LIN {X 0,Y 331.861,Z 837.829,A -85,B 0,C 180,E1 -14617.89,E2 -14617.89} C_VEL
LIN {X 0,Y 331.677,Z 838.758,A -85,B 0,C 180,E1 -14620.289,E2 -14620.289} C_VEL
LIN {X 0,Y 331.646,Z 838.125,A -85,B 0,C 180,E1 -14622.697,E2 -14622.697} C_VEL
LIN {X 0,Y 331.773,Z 836.768,A -85,B 0,C 180,E1 -14624.35,E2 -14624.35} C_VEL
LIN {X 0,Y 332.117,Z 833.423,A -85,B 0,C 180,E1 -14626.716,E2 -14626.716} C_VEL
LIN {X 0,Y 332.464,Z 829.979,A -85,B 0,C 180,E1 -14628.415,E2 -14628.415} C_VEL
LIN {X 0,Y 332.932,Z 825.524,A -85,B 0,C 180,E1 -14630.123,E2 -14630.123} C_VEL
LIN {X 0,Y 333.677,Z 818.981,A -85,B 0,C 180,E1 -14632.096,E2 -14632.096} C_VEL
LIN {X 0,Y 334.531,Z 811.128,A -85,B 0,C 180,E1 -14633.969,E2 -14633.969} C_VEL
LIN {X 0,Y 335.575,Z 802.763,A -85,B 0,C 180,E1 -14635.567,E2 -14635.567} C_VEL
LIN {X 0,Y 336.737,Z 792.663,A -85,B 0,C 180,E1 -14637.137,E2 -14637.137} C_VEL
LIN {X 0,Y 337.93,Z 781.617,A -85,B 0,C 180,E1 -14638.505,E2 -14638.505} C_VEL
LIN {X 0,Y 339.094,Z 769.813,A -85,B 0,C 180,E1 -14639.657,E2 -14639.657} C_VEL
LIN {X 0,Y 339.897,Z 760.336,A -85,B 0,C 180,E1 -14640.387,E2 -14640.387} C_VEL
LIN {X 0,Y 338.213,Z 747.883,A -85,B 0,C 180,E1 -14641.264,E2 -14641.264} C_VEL
LIN {X 0,Y 335.724,Z 734.171,A -85,B 0,C 180,E1 -14641.988,E2 -14641.988} C_VEL
LIN {X 0,Y 334.799,Z 729.351,A -85,B 0,C 180,E1 -14642.208,E2 -14642.208} C_VEL
LIN {X 0,Y 335.382,Z 720.343,A -85,B 0,C 180,E1 -14645.223,E2 -14645.223} C_VEL
LIN {X 0,Y 336.06,Z 710.471,A -85,B 0,C 180,E1 -14648.533,E2 -14648.533} C_VEL
LIN {X 0,Y 336.777,Z 699.019,A -85,B 0,C 180,E1 -14652.387,E2 -14652.387} C_VEL
LIN {X 0,Y 337.478,Z 687.894,A -85,B 0,C 180,E1 -14656.144,E2 -14656.144} C_VEL
LIN {X 0,Y 337.713,Z 680.208,A -85,B 0,C 180,E1 -14658.774,E2 -14658.774} C_VEL
LIN {X 0,Y 336.611,Z 672.395,A -85,B 0,C 180,E1 -14661.597,E2 -14661.597} C_VEL
LIN {X 0,Y 335.43,Z 665.891,A -85,B 0,C 180,E1 -14663.987,E2 -14663.987} C_VEL
LIN {X 0,Y 333.91,Z 658.899,A -85,B 0,C 180,E1 -14666.682,E2 -14666.682} C_VEL
LIN {X 0,Y 334.089,Z 658.875,A -85,B 0,C 180,E1 -14668.795,E2 -14668.795} C_VEL
LIN {X 0,Y 334.249,Z 658.852,A -85,B 0,C 180,E1 -14670.001,E2 -14670.001} C_VEL
LIN {X 0,Y 334.133,Z 658.866,A -85,B 0,C 180,E1 -14672.412,E2 -14672.412} C_VEL
LIN {X 0,Y 334.014,Z 658.877,A -85,B 0,C 180,E1 -14677.253,E2 -14677.253} C_VEL
LIN {X 0,Y 333.839,Z 658.9,A -85,B 0,C 180,E1 -14680.922,E2 -14680.922} C_VEL
LIN {X 0,Y 333.81,Z 658.906,A -85,B 0,C 180,E1 -14684.635,E2 -14684.635} C_VEL
LIN {X 0,Y 333.799,Z 658.91,A -85,B 0,C 180,E1 -14687.816,E2 -14687.816} C_VEL
LIN {X 0,Y 337.948,Z 672.337,A -85,B 0,C 180,E1 -14689.075,E2 -14689.075} C_VEL
LIN {X 0,Y 340.518,Z 682.415,A -85,B 0,C 180,E1 -14690.207,E2 -14690.207} C_VEL
LIN {X 0,Y 339.514,Z 694.142,A -85,B 0,C 180,E1 -14691.559,E2 -14691.559} C_VEL
LIN {X 0,Y 338.525,Z 704.562,A -85,B 0,C 180,E1 -14693.071,E2 -14693.071} C_VEL
LIN {X 0,Y 337.574,Z 713.136,A -85,B 0,C 180,E1 -14694.607,E2 -14694.607} C_VEL
LIN {X 0,Y 336.576,Z 721.162,A -85,B 0,C 180,E1 -14696.368,E2 -14696.368} C_VEL
LIN {X 0,Y 335.902,Z 726.882,A -85,B 0,C 180,E1 -14697.91,E2 -14697.91} C_VEL
LIN {X 0,Y 335.263,Z 731.79,A -85,B 0,C 180,E1 -14699.514,E2 -14699.514} C_VEL
LIN {X 0,Y 334.713,Z 736.907,A -85,B 0,C 180,E1 -14701.664,E2 -14701.664} C_VEL
LIN {X 0,Y 334.206,Z 740.618,A -85,B 0,C 180,E1 -14703.867,E2 -14703.867} C_VEL
LIN {X 0,Y 333.934,Z 742.948,A -85,B 0,C 180,E1 -14706.107,E2 -14706.107} C_VEL
LIN {X 0,Y 333.914,Z 743.791,A -85,B 0,C 180,E1 -14707.857,E2 -14707.857} C_VEL
LIN {X 0,Y 334.024,Z 743.924,A -85,B 0,C 180,E1 -14709.14,E2 -14709.14} C_VEL
LIN {X 0,Y 334.202,Z 743.41,A -85,B 0,C 180,E1 -14710.795,E2 -14710.795} C_VEL
LIN {X 0,Y 334.556,Z 741.933,A -85,B 0,C 180,E1 -14712.672,E2 -14712.672} C_VEL
LIN {X 0,Y 334.657,Z 741.434,A -85,B 0,C 180,E1 -14713.083,E2 -14713.083} C_VEL
LIN {X 0,Y 334.288,Z 740.325,A -85,B 0,C 180,E1 -14714.071,E2 -14714.071} C_VEL
LIN {X 0,Y 332.022,Z 738.157,A -85,B 0,C 180,E1 -14715.689,E2 -14715.689} C_VEL
LIN {X 0,Y 329.839,Z 735.369,A -85,B 0,C 180,E1 -14717.297,E2 -14717.297} C_VEL
LIN {X 0,Y 329.61,Z 733.111,A -85,B 0,C 180,E1 -14718.253,E2 -14718.253} C_VEL
LIN {X 0,Y 330.871,Z 726.379,A -85,B 0,C 180,E1 -14720.415,E2 -14720.415} C_VEL
LIN {X 0,Y 332.059,Z 719.549,A -85,B 0,C 180,E1 -14722.137,E2 -14722.137} C_VEL
LIN {X 0,Y 333.257,Z 711.36,A -85,B 0,C 180,E1 -14723.809,E2 -14723.809} C_VEL
LIN {X 0,Y 334.746,Z 701.133,A -85,B 0,C 180,E1 -14725.468,E2 -14725.468} C_VEL
LIN {X 0,Y 335.956,Z 690.893,A -85,B 0,C 180,E1 -14726.802,E2 -14726.802} C_VEL
LIN {X 0,Y 336.267,Z 687.695,A -85,B 0,C 180,E1 -14727.159,E2 -14727.159} C_VEL
LIN {X 0,Y 333.454,Z 677.696,A -85,B 0,C 180,E1 -14728.469,E2 -14728.469} C_VEL
LIN {X 0,Y 329.206,Z 666.464,A -85,B 0,C 180,E1 -14729.785,E2 -14729.785} C_VEL
LIN {X 0,Y 326.661,Z 659.793,A -85,B 0,C 180,E1 -14730.474,E2 -14730.474} C_VEL
LIN {X 0,Y 326.691,Z 659.789,A -85,B 0,C 180,E1 -14734.517,E2 -14734.517} C_VEL
LIN {X 0,Y 326.623,Z 659.802,A -85,B 0,C 180,E1 -14738.544,E2 -14738.544} C_VEL
LIN {X 0,Y 326.746,Z 659.786,A -85,B 0,C 180,E1 -14741.178,E2 -14741.178} C_VEL
LIN {X 0,Y 326.765,Z 659.781,A -85,B 0,C 180,E1 -14745.433,E2 -14745.433} C_VEL
LIN {X 0,Y 326.771,Z 659.775,A -85,B 0,C 180,E1 -14748.839,E2 -14748.839} C_VEL
LIN {X 0,Y 326.981,Z 659.745,A -85,B 0,C 180,E1 -14752.591,E2 -14752.591} C_VEL
LIN {X 0,Y 326.78,Z 659.778,A -85,B 0,C 180,E1 -14755.065,E2 -14755.065} C_VEL
LIN {X 0,Y 327.049,Z 659.738,A -85,B 0,C 180,E1 -14757.537,E2 -14757.537} C_VEL
LIN {X 0,Y 327.2,Z 659.721,A -85,B 0,C 180,E1 -14760,E2 -14760} C_VEL
LIN {X 0,Y 327.05,Z 659.746,A -85,B 0,C 180,E1 -14762.463,E2 -14762.463} C_VEL
LIN {X 0,Y 326.998,Z 659.748,A -85,B 0,C 180,E1 -14766.169,E2 -14766.169} C_VEL
LIN {X 0,Y 326.917,Z 659.754,A -85,B 0,C 180,E1 -14768.655,E2 -14768.655} C_VEL
LIN {X 0,Y 326.736,Z 659.779,A -85,B 0,C 180,E1 -14772.421,E2 -14772.421} C_VEL
LIN {X 0,Y 326.756,Z 659.782,A -85,B 0,C 180,E1 -14774.958,E2 -14774.958} C_VEL
LIN {X 0,Y 326.736,Z 659.783,A -85,B 0,C 180,E1 -14778.839,E2 -14778.839} C_VEL
LIN {X 0,Y 326.623,Z 659.794,A -85,B 0,C 180,E1 -14782.787,E2 -14782.787} C_VEL
LIN {X 0,Y 326.692,Z 659.787,A -85,B 0,C 180,E1 -14785.484,E2 -14785.484} C_VEL
LIN {X 0,Y 326.65,Z 659.797,A -85,B 0,C 180,E1 -14789.66,E2 -14789.66} C_VEL
LIN {X 0,Y 326.609,Z 659.805,A -85,B 0,C 180,E1 -14794.019,E2 -14794.019} C_VEL
LIN {X 0,Y 326.63,Z 659.803,A -85,B 0,C 180,E1 -14797.239,E2 -14797.239} C_VEL
LIN {X 0,Y 326.629,Z 659.853,A -85,B 0,C 180,E1 -14800.58,E2 -14800.58} C_VEL
LIN {X 0,Y 328.011,Z 666.445,A -85,B 0,C 180,E1 -14804.135,E2 -14804.135} C_VEL
LIN {X 0,Y 329.365,Z 673.292,A -85,B 0,C 180,E1 -14807.488,E2 -14807.488} C_VEL
LIN {X 0,Y 330.58,Z 679.663,A -85,B 0,C 180,E1 -14810.372,E2 -14810.372} C_VEL
LIN {X 0,Y 331.086,Z 683.496,A -85,B 0,C 180,E1 -14812.005,E2 -14812.005} C_VEL
LIN {X 0,Y 330.051,Z 691.01,A -85,B 0,C 180,E1 -14814.905,E2 -14814.905} C_VEL
LIN {X 0,Y 328.741,Z 701.452,A -85,B 0,C 180,E1 -14818.776,E2 -14818.776} C_VEL
LIN {X 0,Y 327.667,Z 711.906,A -85,B 0,C 180,E1 -14822.538,E2 -14822.538} C_VEL
LIN {X 0,Y 326.622,Z 724.408,A -85,B 0,C 180,E1 -14826.853,E2 -14826.853} C_VEL
LIN {X 0,Y 329.145,Z 739.18,A -85,B 0,C 180,E1 -14827.642,E2 -14827.642} C_VEL
LIN {X 0,Y 330.443,Z 751.644,A -85,B 0,C 180,E1 -14828.469,E2 -14828.469} C_VEL
LIN {X 0,Y 331.025,Z 765.509,A -85,B 0,C 180,E1 -14829.568,E2 -14829.568} C_VEL
LIN {X 0,Y 331.436,Z 777.667,A -85,B 0,C 180,E1 -14830.328,E2 -14830.328} C_VEL
LIN {X 0,Y 331.574,Z 787.793,A -85,B 0,C 180,E1 -14831.141,E2 -14831.141} C_VEL
LIN {X 0,Y 330.277,Z 800.215,A -85,B 0,C 180,E1 -14832.348,E2 -14832.348} C_VEL
LIN {X 0,Y 329.137,Z 811.195,A -85,B 0,C 180,E1 -14833.724,E2 -14833.724} C_VEL
LIN {X 0,Y 328.186,Z 820.112,A -85,B 0,C 180,E1 -14835.109,E2 -14835.109} C_VEL
LIN {X 0,Y 327.013,Z 829.783,A -85,B 0,C 180,E1 -14836.958,E2 -14836.958} C_VEL
LIN {X 0,Y 326.136,Z 837.451,A -85,B 0,C 180,E1 -14838.816,E2 -14838.816} C_VEL
LIN {X 0,Y 325.595,Z 843.592,A -85,B 0,C 180,E1 -14840.683,E2 -14840.683} C_VEL
LIN {X 0,Y 325.224,Z 848.431,A -85,B 0,C 180,E1 -14842.55,E2 -14842.55} C_VEL
LIN {X 0,Y 325.077,Z 851.374,A -85,B 0,C 180,E1 -14843.988,E2 -14843.988} C_VEL
LIN {X 0,Y 324.996,Z 854.734,A -85,B 0,C 180,E1 -14846.28,E2 -14846.28} C_VEL
LIN {X 0,Y 324.927,Z 855.95,A -85,B 0,C 180,E1 -14847.52,E2 -14847.52} C_VEL
LIN {X 0,Y 324.959,Z 856.716,A -85,B 0,C 180,E1 -14848.76,E2 -14848.76} C_VEL
LIN {X 0,Y 325.011,Z 857.06,A -85,B 0,C 180,E1 -14849.999,E2 -14849.999} C_VEL
LIN {X 0,Y 324.942,Z 857.003,A -85,B 0,C 180,E1 -14851.239,E2 -14851.239} C_VEL
LIN {X 0,Y 324.922,Z 856.543,A -85,B 0,C 180,E1 -14852.479,E2 -14852.479} C_VEL
LIN {X 0,Y 324.987,Z 855.631,A -85,B 0,C 180,E1 -14853.719,E2 -14853.719} C_VEL
LIN {X 0,Y 325.018,Z 853.014,A -85,B 0,C 180,E1 -14855.912,E2 -14855.912} C_VEL
LIN {X 0,Y 325.344,Z 849.12,A -85,B 0,C 180,E1 -14858.071,E2 -14858.071} C_VEL
LIN {X 0,Y 325.842,Z 844.566,A -85,B 0,C 180,E1 -14859.935,E2 -14859.935} C_VEL
LIN {X 0,Y 326.665,Z 837.655,A -85,B 0,C 180,E1 -14862.108,E2 -14862.108} C_VEL
LIN {X 0,Y 327.841,Z 830.181,A -85,B 0,C 180,E1 -14863.955,E2 -14863.955} C_VEL
LIN {X 0,Y 328.887,Z 822.723,A -85,B 0,C 180,E1 -14865.465,E2 -14865.465} C_VEL
LIN {X 0,Y 330.233,Z 813.387,A -85,B 0,C 180,E1 -14867.014,E2 -14867.014} C_VEL
LIN {X 0,Y 331.627,Z 803.213,A -85,B 0,C 180,E1 -14868.374,E2 -14868.374} C_VEL
LIN {X 0,Y 333.125,Z 792.076,A -85,B 0,C 180,E1 -14869.567,E2 -14869.567} C_VEL
LIN {X 0,Y 333.537,Z 783.566,A -85,B 0,C 180,E1 -14870.344,E2 -14870.344} C_VEL
LIN {X 0,Y 333.449,Z 770.917,A -85,B 0,C 180,E1 -14871.311,E2 -14871.311} C_VEL
LIN {X 0,Y 332.694,Z 757.681,A -85,B 0,C 180,E1 -14872.083,E2 -14872.083} C_VEL
LIN {X 0,Y 330.545,Z 744.372,A -85,B 0,C 180,E1 -14872.731,E2 -14872.731} C_VEL
LIN {X 0,Y 329.17,Z 737.997,A -85,B 0,C 180,E1 -14873.061,E2 -14873.061} C_VEL
LIN {X 0,Y 327.482,Z 722.292,A -85,B 0,C 180,E1 -14874.907,E2 -14874.907} C_VEL
LIN {X 0,Y 327.209,Z 718.727,A -85,B 0,C 180,E1 -14875.354,E2 -14875.354} C_VEL
LIN {X 0,Y 328.159,Z 708.48,A -85,B 0,C 180,E1 -14878.967,E2 -14878.967} C_VEL
LIN {X 0,Y 329.462,Z 697.365,A -85,B 0,C 180,E1 -14882.952,E2 -14882.952} C_VEL
LIN {X 0,Y 330.775,Z 687.687,A -85,B 0,C 180,E1 -14886.506,E2 -14886.506} C_VEL
LIN {X 0,Y 331.077,Z 683.113,A -85,B 0,C 180,E1 -14888.24,E2 -14888.24} C_VEL
LIN {X 0,Y 330.054,Z 676.875,A -85,B 0,C 180,E1 -14890.768,E2 -14890.768} C_VEL
LIN {X 0,Y 328.431,Z 668.84,A -85,B 0,C 180,E1 -14894.205,E2 -14894.205} C_VEL
LIN {X 0,Y 326.669,Z 659.795,A -85,B 0,C 180,E1 -14898.317,E2 -14898.317} C_VEL
LIN {X 0,Y 326.644,Z 659.797,A -85,B 0,C 180,E1 -14901.394,E2 -14901.394} C_VEL
LIN {X 0,Y 326.616,Z 659.795,A -85,B 0,C 180,E1 -14904.85,E2 -14904.85} C_VEL
LIN {X 0,Y 326.604,Z 659.8,A -85,B 0,C 180,E1 -14907.455,E2 -14907.455} C_VEL
LIN {X 0,Y 326.657,Z 659.794,A -85,B 0,C 180,E1 -14910.34,E2 -14910.34} C_VEL
LIN {X 0,Y 326.686,Z 659.785,A -85,B 0,C 180,E1 -14914.516,E2 -14914.516} C_VEL
LIN {X 0,Y 326.645,Z 659.798,A -85,B 0,C 180,E1 -14918.545,E2 -14918.545} C_VEL
LIN {X 0,Y 326.74,Z 659.787,A -85,B 0,C 180,E1 -14921.177,E2 -14921.177} C_VEL
LIN {X 0,Y 326.758,Z 659.781,A -85,B 0,C 180,E1 -14925.433,E2 -14925.433} C_VEL
LIN {X 0,Y 326.769,Z 659.78,A -85,B 0,C 180,E1 -14928.839,E2 -14928.839} C_VEL
LIN {X 0,Y 326.964,Z 659.839,A -85,B 0,C 180,E1 -14932.071,E2 -14932.071} C_VEL
LIN {X 0,Y 328.395,Z 665.268,A -85,B 0,C 180,E1 -14934.473,E2 -14934.473} C_VEL
LIN {X 0,Y 330.562,Z 672.965,A -85,B 0,C 180,E1 -14937.762,E2 -14937.762} C_VEL
LIN {X 0,Y 331.697,Z 678.579,A -85,B 0,C 180,E1 -14940,E2 -14940} C_VEL
LIN {X 0,Y 332.394,Z 684.908,A -85,B 0,C 180,E1 -14942.423,E2 -14942.423} C_VEL
LIN {X 0,Y 332.288,Z 690.153,A -85,B 0,C 180,E1 -14944.245,E2 -14944.245} C_VEL
LIN {X 0,Y 331.442,Z 699.025,A -85,B 0,C 180,E1 -14947.309,E2 -14947.309} C_VEL
LIN {X 0,Y 330.633,Z 710.037,A -85,B 0,C 180,E1 -14951.029,E2 -14951.029} C_VEL
LIN {X 0,Y 329.691,Z 721.175,A -85,B 0,C 180,E1 -14954.821,E2 -14954.821} C_VEL
LIN {X 0,Y 329.004,Z 730.381,A -85,B 0,C 180,E1 -14957.963,E2 -14957.963} C_VEL
LIN {X 0,Y 332.669,Z 744.629,A -85,B 0,C 180,E1 -14958.874,E2 -14958.874} C_VEL
LIN {X 0,Y 334.735,Z 756.733,A -85,B 0,C 180,E1 -14959.789,E2 -14959.789} C_VEL
LIN {X 0,Y 335.355,Z 762.9,A -85,B 0,C 180,E1 -14960.31,E2 -14960.31} C_VEL
LIN {X 0,Y 334.182,Z 773.988,A -85,B 0,C 180,E1 -14961.24,E2 -14961.24} C_VEL
LIN {X 0,Y 332.896,Z 784.331,A -85,B 0,C 180,E1 -14962.334,E2 -14962.334} C_VEL
LIN {X 0,Y 331.359,Z 795.104,A -85,B 0,C 180,E1 -14963.765,E2 -14963.765} C_VEL
LIN {X 0,Y 330,Z 803.961,A -85,B 0,C 180,E1 -14965.21,E2 -14965.21} C_VEL
LIN {X 0,Y 328.635,Z 812.956,A -85,B 0,C 180,E1 -14967.029,E2 -14967.029} C_VEL
LIN {X 0,Y 327.396,Z 820.622,A -85,B 0,C 180,E1 -14968.983,E2 -14968.983} C_VEL
LIN {X 0,Y 326.65,Z 825.766,A -85,B 0,C 180,E1 -14970.616,E2 -14970.616} C_VEL
LIN {X 0,Y 325.833,Z 831.035,A -85,B 0,C 180,E1 -14972.735,E2 -14972.735} C_VEL
LIN {X 0,Y 325.256,Z 834.796,A -85,B 0,C 180,E1 -14974.808,E2 -14974.808} C_VEL
LIN {X 0,Y 324.882,Z 837.267,A -85,B 0,C 180,E1 -14976.833,E2 -14976.833} C_VEL
LIN {X 0,Y 324.681,Z 838.649,A -85,B 0,C 180,E1 -14978.883,E2 -14978.883} C_VEL
LIN {X 0,Y 324.561,Z 838.967,A -85,B 0,C 180,E1 -14980.724,E2 -14980.724} C_VEL
LIN {X 0,Y 324.544,Z 838.382,A -85,B 0,C 180,E1 -14982.587,E2 -14982.587} C_VEL
LIN {X 0,Y 324.681,Z 836.911,A -85,B 0,C 180,E1 -14984.414,E2 -14984.414} C_VEL
LIN {X 0,Y 324.929,Z 834.578,A -85,B 0,C 180,E1 -14986.202,E2 -14986.202} C_VEL
LIN {X 0,Y 325.274,Z 831.396,A -85,B 0,C 180,E1 -14987.95,E2 -14987.95} C_VEL
LIN {X 0,Y 325.664,Z 827.371,A -85,B 0,C 180,E1 -14989.654,E2 -14989.654} C_VEL
LIN {X 0,Y 326.418,Z 821.17,A -85,B 0,C 180,E1 -14991.711,E2 -14991.711} C_VEL
LIN {X 0,Y 327.195,Z 814.686,A -85,B 0,C 180,E1 -14993.413,E2 -14993.413} C_VEL
LIN {X 0,Y 328.28,Z 806.003,A -85,B 0,C 180,E1 -14995.251,E2 -14995.251} C_VEL
LIN {X 0,Y 329.425,Z 796.379,A -85,B 0,C 180,E1 -14996.895,E2 -14996.895} C_VEL
LIN {X 0,Y 330.744,Z 784.873,A -85,B 0,C 180,E1 -14998.451,E2 -14998.451} C_VEL
LIN {X 0,Y 331.965,Z 772.941,A -85,B 0,C 180,E1 -14999.719,E2 -14999.719} C_VEL
LIN {X 0,Y 333.047,Z 761.183,A -85,B 0,C 180,E1 -15000.68,E2 -15000.68} C_VEL
LIN {X 0,Y 331.507,Z 749.49,A -85,B 0,C 180,E1 -15001.54,E2 -15001.54} C_VEL
LIN {X 0,Y 329.18,Z 736.298,A -85,B 0,C 180,E1 -15002.289,E2 -15002.289} C_VEL
LIN {X 0,Y 327.875,Z 729.497,A -85,B 0,C 180,E1 -15002.602,E2 -15002.602} C_VEL
LIN {X 0,Y 328.521,Z 719.419,A -85,B 0,C 180,E1 -15006.018,E2 -15006.018} C_VEL
LIN {X 0,Y 329.272,Z 709.539,A -85,B 0,C 180,E1 -15009.381,E2 -15009.381} C_VEL
LIN {X 0,Y 329.965,Z 698.474,A -85,B 0,C 180,E1 -15013.146,E2 -15013.146} C_VEL
LIN {X 0,Y 330.589,Z 688.749,A -85,B 0,C 180,E1 -15016.477,E2 -15016.477} C_VEL
LIN {X 0,Y 330.821,Z 681.535,A -85,B 0,C 180,E1 -15018.978,E2 -15018.978} C_VEL
LIN {X 0,Y 329.618,Z 673.201,A -85,B 0,C 180,E1 -15022.034,E2 -15022.034} C_VEL
LIN {X 0,Y 328.353,Z 666.71,A -85,B 0,C 180,E1 -15024.474,E2 -15024.474} C_VEL
LIN {X 0,Y 326.946,Z 659.765,A -85,B 0,C 180,E1 -15027.151,E2 -15027.151} C_VEL
LIN {X 0,Y 327.2,Z 659.729,A -85,B 0,C 180,E1 -15030.001,E2 -15030.001} C_VEL
LIN {X 0,Y 327.069,Z 659.746,A -85,B 0,C 180,E1 -15032.464,E2 -15032.464} C_VEL
LIN {X 0,Y 326.992,Z 659.751,A -85,B 0,C 180,E1 -15036.17,E2 -15036.17} C_VEL
LIN {X 0,Y 326.916,Z 659.764,A -85,B 0,C 180,E1 -15038.656,E2 -15038.656} C_VEL
LIN {X 0,Y 326.74,Z 659.785,A -85,B 0,C 180,E1 -15042.422,E2 -15042.422} C_VEL
LIN {X 0,Y 326.756,Z 659.785,A -85,B 0,C 180,E1 -15044.958,E2 -15044.958} C_VEL
LIN {X 0,Y 326.765,Z 659.96,A -85,B 0,C 180,E1 -15047.444,E2 -15047.444} C_VEL
LIN {X 0,Y 330.61,Z 672.1,A -85,B 0,C 180,E1 -15048.595,E2 -15048.595} C_VEL
LIN {X 0,Y 333.671,Z 683.136,A -85,B 0,C 180,E1 -15049.855,E2 -15049.855} C_VEL
LIN {X 0,Y 332.849,Z 693.349,A -85,B 0,C 180,E1 -15051.036,E2 -15051.036} C_VEL
LIN {X 0,Y 331.82,Z 704.103,A -85,B 0,C 180,E1 -15052.575,E2 -15052.575} C_VEL
LIN {X 0,Y 330.804,Z 713.337,A -85,B 0,C 180,E1 -15054.217,E2 -15054.217} C_VEL
LIN {X 0,Y 329.689,Z 721.838,A -85,B 0,C 180,E1 -15056.095,E2 -15056.095} C_VEL
LIN {X 0,Y 328.804,Z 728.896,A -85,B 0,C 180,E1 -15058.05,E2 -15058.05} C_VEL
LIN {X 0,Y 328.258,Z 733.106,A -85,B 0,C 180,E1 -15059.501,E2 -15059.501} C_VEL
LIN {X 0,Y 327.677,Z 738.165,A -85,B 0,C 180,E1 -15061.7,E2 -15061.7} C_VEL
LIN {X 0,Y 327.172,Z 741.793,A -85,B 0,C 180,E1 -15063.953,E2 -15063.953} C_VEL
LIN {X 0,Y 326.967,Z 743.479,A -85,B 0,C 180,E1 -15065.476,E2 -15065.476} C_VEL
LIN {X 0,Y 326.878,Z 744.654,A -85,B 0,C 180,E1 -15067.296,E2 -15067.296} C_VEL
LIN {X 0,Y 327.014,Z 744.962,A -85,B 0,C 180,E1 -15069.314,E2 -15069.314} C_VEL
LIN {X 0,Y 327.352,Z 743.951,A -85,B 0,C 180,E1 -15071.725,E2 -15071.725} C_VEL
LIN {X 0,Y 327.976,Z 741.402,A -85,B 0,C 180,E1 -15074.141,E2 -15074.141} C_VEL
LIN {X 0,Y 328.544,Z 738.73,A -85,B 0,C 180,E1 -15075.775,E2 -15075.775} C_VEL
LIN {X 0,Y 329.298,Z 735.012,A -85,B 0,C 180,E1 -15077.504,E2 -15077.504} C_VEL
LIN {X 0,Y 329.61,Z 733.111,A -85,B 0,C 180,E1 -15078.253,E2 -15078.253} C_VEL
LIN {X 0,Y 329.429,Z 730.708,A -85,B 0,C 180,E1 -15079.193,E2 -15079.193} C_VEL
LIN {X 0,Y 327.534,Z 726.522,A -85,B 0,C 180,E1 -15080.727,E2 -15080.727} C_VEL
LIN {X 0,Y 325.754,Z 721.651,A -85,B 0,C 180,E1 -15082.207,E2 -15082.207} C_VEL
LIN {X 0,Y 325.739,Z 718.164,A -85,B 0,C 180,E1 -15083.045,E2 -15083.045} C_VEL
LIN {X 0,Y 327.099,Z 709.512,A -85,B 0,C 180,E1 -15084.733,E2 -15084.733} C_VEL
LIN {X 0,Y 328.472,Z 700.088,A -85,B 0,C 180,E1 -15086.2,E2 -15086.2} C_VEL
LIN {X 0,Y 329.624,Z 689.263,A -85,B 0,C 180,E1 -15087.572,E2 -15087.572} C_VEL
LIN {X 0,Y 326.796,Z 679.346,A -85,B 0,C 180,E1 -15088.927,E2 -15088.927} C_VEL
LIN {X 0,Y 323.09,Z 669.418,A -85,B 0,C 180,E1 -15090.16,E2 -15090.16} C_VEL
LIN {X 0,Y 319.683,Z 661.004,A -85,B 0,C 180,E1 -15091.076,E2 -15091.076} C_VEL
LIN {X 0,Y 319.611,Z 660.671,A -85,B 0,C 180,E1 -15091.15,E2 -15091.15} C_VEL
LIN {X 0,Y 319.605,Z 660.675,A -85,B 0,C 180,E1 -15095.304,E2 -15095.304} C_VEL
LIN {X 0,Y 319.606,Z 660.678,A -85,B 0,C 180,E1 -15099.401,E2 -15099.401} C_VEL
LIN {X 0,Y 319.66,Z 660.669,A -85,B 0,C 180,E1 -15102.073,E2 -15102.073} C_VEL
LIN {X 0,Y 319.734,Z 660.657,A -85,B 0,C 180,E1 -15106.008,E2 -15106.008} C_VEL
LIN {X 0,Y 319.76,Z 660.654,A -85,B 0,C 180,E1 -15109.873,E2 -15109.873} C_VEL
LIN {X 0,Y 319.935,Z 660.623,A -85,B 0,C 180,E1 -15112.426,E2 -15112.426} C_VEL
LIN {X 0,Y 319.749,Z 660.654,A -85,B 0,C 180,E1 -15114.956,E2 -15114.956} C_VEL
LIN {X 0,Y 319.993,Z 660.616,A -85,B 0,C 180,E1 -15117.483,E2 -15117.483} C_VEL
LIN {X 0,Y 320.152,Z 660.599,A -85,B 0,C 180,E1 -15120,E2 -15120} C_VEL
LIN {X 0,Y 319.994,Z 660.625,A -85,B 0,C 180,E1 -15122.518,E2 -15122.518} C_VEL
LIN {X 0,Y 319.954,Z 660.627,A -85,B 0,C 180,E1 -15126.306,E2 -15126.306} C_VEL
LIN {X 0,Y 319.845,Z 660.634,A -85,B 0,C 180,E1 -15128.848,E2 -15128.848} C_VEL
LIN {X 0,Y 319.683,Z 660.656,A -85,B 0,C 180,E1 -15132.7,E2 -15132.7} C_VEL
LIN {X 0,Y 319.702,Z 660.66,A -85,B 0,C 180,E1 -15135.296,E2 -15135.296} C_VEL
LIN {X 0,Y 319.677,Z 660.661,A -85,B 0,C 180,E1 -15139.255,E2 -15139.255} C_VEL
LIN {X 0,Y 319.572,Z 660.673,A -85,B 0,C 180,E1 -15143.319,E2 -15143.319} C_VEL
LIN {X 0,Y 319.62,Z 660.668,A -85,B 0,C 180,E1 -15146.09,E2 -15146.09} C_VEL
LIN {X 0,Y 319.582,Z 660.676,A -85,B 0,C 180,E1 -15148.935,E2 -15148.935} C_VEL
LIN {X 0,Y 319.533,Z 660.685,A -85,B 0,C 180,E1 -15151.862,E2 -15151.862} C_VEL
LIN {X 0,Y 319.582,Z 660.68,A -85,B 0,C 180,E1 -15155.543,E2 -15155.543} C_VEL
LIN {X 0,Y 319.561,Z 660.681,A -85,B 0,C 180,E1 -15159.669,E2 -15159.669} C_VEL
LIN {X 0,Y 319.608,Z 660.998,A -85,B 0,C 180,E1 -15160.03,E2 -15160.03} C_VEL
LIN {X 0,Y 321.03,Z 667.662,A -85,B 0,C 180,E1 -15163.743,E2 -15163.743} C_VEL
LIN {X 0,Y 322.241,Z 673.623,A -85,B 0,C 180,E1 -15166.785,E2 -15166.785} C_VEL
LIN {X 0,Y 323.64,Z 681.063,A -85,B 0,C 180,E1 -15170.273,E2 -15170.273} C_VEL
LIN {X 0,Y 324.106,Z 685.046,A -85,B 0,C 180,E1 -15171.989,E2 -15171.989} C_VEL
LIN {X 0,Y 322.806,Z 693.983,A -85,B 0,C 180,E1 -15175.523,E2 -15175.523} C_VEL
LIN {X 0,Y 321.57,Z 703.448,A -85,B 0,C 180,E1 -15179.1,E2 -15179.1} C_VEL
LIN {X 0,Y 320.579,Z 712.936,A -85,B 0,C 180,E1 -15182.588,E2 -15182.588} C_VEL
LIN {X 0,Y 319.667,Z 723.025,A -85,B 0,C 180,E1 -15186.199,E2 -15186.199} C_VEL
LIN {X 0,Y 322.369,Z 738.671,A -85,B 0,C 180,E1 -15187.086,E2 -15187.086} C_VEL
LIN {X 0,Y 323.668,Z 751.03,A -85,B 0,C 180,E1 -15187.951,E2 -15187.951} C_VEL
LIN {X 0,Y 324.164,Z 764.057,A -85,B 0,C 180,E1 -15189.065,E2 -15189.065} C_VEL
LIN {X 0,Y 324.323,Z 770.273,A -85,B 0,C 180,E1 -15189.474,E2 -15189.474} C_VEL
LIN {X 0,Y 324.702,Z 782.978,A -85,B 0,C 180,E1 -15190.397,E2 -15190.397} C_VEL
LIN {X 0,Y 324.537,Z 790.321,A -85,B 0,C 180,E1 -15191.044,E2 -15191.044} C_VEL
LIN {X 0,Y 323.319,Z 800.819,A -85,B 0,C 180,E1 -15192.119,E2 -15192.119} C_VEL
LIN {X 0,Y 322.143,Z 811.603,A -85,B 0,C 180,E1 -15193.523,E2 -15193.523} C_VEL
LIN {X 0,Y 321.054,Z 821.311,A -85,B 0,C 180,E1 -15195.095,E2 -15195.095} C_VEL
LIN {X 0,Y 320.074,Z 829.268,A -85,B 0,C 180,E1 -15196.67,E2 -15196.67} C_VEL
LIN {X 0,Y 319.114,Z 837.012,A -85,B 0,C 180,E1 -15198.567,E2 -15198.567} C_VEL
LIN {X 0,Y 318.551,Z 843.2,A -85,B 0,C 180,E1 -15200.475,E2 -15200.475} C_VEL
LIN {X 0,Y 318.177,Z 848.081,A -85,B 0,C 180,E1 -15202.384,E2 -15202.384} C_VEL
LIN {X 0,Y 317.97,Z 851.405,A -85,B 0,C 180,E1 -15204.057,E2 -15204.057} C_VEL
LIN {X 0,Y 317.902,Z 854.458,A -85,B 0,C 180,E1 -15206.197,E2 -15206.197} C_VEL
LIN {X 0,Y 317.846,Z 855.692,A -85,B 0,C 180,E1 -15207.465,E2 -15207.465} C_VEL
LIN {X 0,Y 317.864,Z 856.49,A -85,B 0,C 180,E1 -15208.732,E2 -15208.732} C_VEL
LIN {X 0,Y 317.913,Z 856.85,A -85,B 0,C 180,E1 -15209.999,E2 -15209.999} C_VEL
LIN {X 0,Y 317.848,Z 856.809,A -85,B 0,C 180,E1 -15211.266,E2 -15211.266} C_VEL
LIN {X 0,Y 317.841,Z 856.372,A -85,B 0,C 180,E1 -15212.534,E2 -15212.534} C_VEL
LIN {X 0,Y 317.892,Z 855.49,A -85,B 0,C 180,E1 -15213.802,E2 -15213.802} C_VEL
LIN {X 0,Y 317.923,Z 853.182,A -85,B 0,C 180,E1 -15215.86,E2 -15215.86} C_VEL
LIN {X 0,Y 318.284,Z 849.059,A -85,B 0,C 180,E1 -15218.251,E2 -15218.251} C_VEL
LIN {X 0,Y 318.835,Z 844.546,A -85,B 0,C 180,E1 -15220.156,E2 -15220.156} C_VEL
LIN {X 0,Y 319.712,Z 837.702,A -85,B 0,C 180,E1 -15222.375,E2 -15222.375} C_VEL
LIN {X 0,Y 320.934,Z 830.278,A -85,B 0,C 180,E1 -15224.261,E2 -15224.261} C_VEL
LIN {X 0,Y 322.134,Z 821.985,A -85,B 0,C 180,E1 -15225.983,E2 -15225.983} C_VEL
LIN {X 0,Y 323.569,Z 812.681,A -85,B 0,C 180,E1 -15227.539,E2 -15227.539} C_VEL
LIN {X 0,Y 325.071,Z 802.452,A -85,B 0,C 180,E1 -15228.922,E2 -15228.922} C_VEL
LIN {X 0,Y 326.635,Z 791.209,A -85,B 0,C 180,E1 -15230.136,E2 -15230.136} C_VEL
LIN {X 0,Y 326.929,Z 782.576,A -85,B 0,C 180,E1 -15230.939,E2 -15230.939} C_VEL
LIN {X 0,Y 326.907,Z 770.404,A -85,B 0,C 180,E1 -15231.878,E2 -15231.878} C_VEL
LIN {X 0,Y 326.202,Z 757.985,A -85,B 0,C 180,E1 -15232.628,E2 -15232.628} C_VEL
LIN {X 0,Y 324.093,Z 745.01,A -85,B 0,C 180,E1 -15233.303,E2 -15233.303} C_VEL
LIN {X 0,Y 322.568,Z 737.897,A -85,B 0,C 180,E1 -15233.685,E2 -15233.685} C_VEL
LIN {X 0,Y 320.898,Z 720.964,A -85,B 0,C 180,E1 -15235.802,E2 -15235.802} C_VEL
LIN {X 0,Y 320.397,Z 715.96,A -85,B 0,C 180,E1 -15236.528,E2 -15236.528} C_VEL
LIN {X 0,Y 321.458,Z 705.881,A -85,B 0,C 180,E1 -15240.187,E2 -15240.187} C_VEL
LIN {X 0,Y 322.802,Z 695.115,A -85,B 0,C 180,E1 -15244.174,E2 -15244.174} C_VEL
LIN {X 0,Y 324.025,Z 686.58,A -85,B 0,C 180,E1 -15247.394,E2 -15247.394} C_VEL
LIN {X 0,Y 323.992,Z 683.388,A -85,B 0,C 180,E1 -15248.656,E2 -15248.656} C_VEL
LIN {X 0,Y 322.795,Z 676.712,A -85,B 0,C 180,E1 -15251.458,E2 -15251.458} C_VEL
LIN {X 0,Y 321.213,Z 668.768,A -85,B 0,C 180,E1 -15254.96,E2 -15254.96} C_VEL
LIN {X 0,Y 319.622,Z 660.674,A -85,B 0,C 180,E1 -15258.779,E2 -15258.779} C_VEL
LIN {X 0,Y 319.58,Z 660.67,A -85,B 0,C 180,E1 -15262.342,E2 -15262.342} C_VEL
LIN {X 0,Y 319.556,Z 660.672,A -85,B 0,C 180,E1 -15265.123,E2 -15265.123} C_VEL
LIN {X 0,Y 319.566,Z 660.673,A -85,B 0,C 180,E1 -15269.057,E2 -15269.057} C_VEL
LIN {X 0,Y 319.605,Z 660.674,A -85,B 0,C 180,E1 -15272.498,E2 -15272.498} C_VEL
LIN {X 0,Y 319.601,Z 660.672,A -85,B 0,C 180,E1 -15275.303,E2 -15275.303} C_VEL
LIN {X 0,Y 319.593,Z 660.674,A -85,B 0,C 180,E1 -15278.047,E2 -15278.047} C_VEL
LIN {X 0,Y 319.685,Z 660.664,A -85,B 0,C 180,E1 -15280.961,E2 -15280.961} C_VEL
LIN {X 0,Y 319.726,Z 660.656,A -85,B 0,C 180,E1 -15285.275,E2 -15285.275} C_VEL
LIN {X 0,Y 319.755,Z 660.655,A -85,B 0,C 180,E1 -15289.873,E2 -15289.873} C_VEL
LIN {X 0,Y 319.849,Z 660.824,A -85,B 0,C 180,E1 -15290.833,E2 -15290.833} C_VEL
LIN {X 0,Y 321.765,Z 666.854,A -85,B 0,C 180,E1 -15293.73,E2 -15293.73} C_VEL
LIN {X 0,Y 324.013,Z 675.44,A -85,B 0,C 180,E1 -15297.513,E2 -15297.513} C_VEL
LIN {X 0,Y 325.168,Z 681.464,A -85,B 0,C 180,E1 -15300,E2 -15300} C_VEL
LIN {X 0,Y 325.763,Z 686.259,A -85,B 0,C 180,E1 -15301.854,E2 -15301.854} C_VEL
LIN {X 0,Y 325.666,Z 691.21,A -85,B 0,C 180,E1 -15303.712,E2 -15303.712} C_VEL
LIN {X 0,Y 324.834,Z 700.298,A -85,B 0,C 180,E1 -15306.834,E2 -15306.834} C_VEL
LIN {X 0,Y 323.892,Z 711.232,A -85,B 0,C 180,E1 -15310.628,E2 -15310.628} C_VEL
LIN {X 0,Y 323.082,Z 720.501,A -85,B 0,C 180,E1 -15313.844,E2 -15313.844} C_VEL
LIN {X 0,Y 322.241,Z 730.553,A -85,B 0,C 180,E1 -15317.327,E2 -15317.327} C_VEL
LIN {X 0,Y 325.909,Z 744.508,A -85,B 0,C 180,E1 -15318.262,E2 -15318.262} C_VEL
LIN {X 0,Y 327.909,Z 755.347,A -85,B 0,C 180,E1 -15319.11,E2 -15319.11} C_VEL
LIN {X 0,Y 328.821,Z 764.222,A -85,B 0,C 180,E1 -15319.88,E2 -15319.88} C_VEL
LIN {X 0,Y 327.51,Z 775.797,A -85,B 0,C 180,E1 -15320.901,E2 -15320.901} C_VEL
LIN {X 0,Y 325.974,Z 786.926,A -85,B 0,C 180,E1 -15322.153,E2 -15322.153} C_VEL
LIN {X 0,Y 324.416,Z 797.383,A -85,B 0,C 180,E1 -15323.627,E2 -15323.627} C_VEL
LIN {X 0,Y 323.032,Z 805.857,A -85,B 0,C 180,E1 -15325.103,E2 -15325.103} C_VEL
LIN {X 0,Y 321.693,Z 814.012,A -85,B 0,C 180,E1 -15326.851,E2 -15326.851} C_VEL
LIN {X 0,Y 320.395,Z 821.542,A -85,B 0,C 180,E1 -15328.854,E2 -15328.854} C_VEL
LIN {X 0,Y 319.446,Z 827.582,A -85,B 0,C 180,E1 -15330.907,E2 -15330.907} C_VEL
LIN {X 0,Y 318.66,Z 832.395,A -85,B 0,C 180,E1 -15333.064,E2 -15333.064} C_VEL
LIN {X 0,Y 318.092,Z 835.787,A -85,B 0,C 180,E1 -15335.168,E2 -15335.168} C_VEL
LIN {X 0,Y 317.753,Z 837.956,A -85,B 0,C 180,E1 -15337.229,E2 -15337.229} C_VEL
LIN {X 0,Y 317.554,Z 839.022,A -85,B 0,C 180,E1 -15339.232,E2 -15339.232} C_VEL
LIN {X 0,Y 317.44,Z 838.982,A -85,B 0,C 180,E1 -15341.62,E2 -15341.62} C_VEL
LIN {X 0,Y 317.49,Z 838.073,A -85,B 0,C 180,E1 -15343.331,E2 -15343.331} C_VEL
LIN {X 0,Y 317.792,Z 835.26,A -85,B 0,C 180,E1 -15345.905,E2 -15345.905} C_VEL
LIN {X 0,Y 318.132,Z 832.278,A -85,B 0,C 180,E1 -15347.684,E2 -15347.684} C_VEL
LIN {X 0,Y 318.642,Z 827.361,A -85,B 0,C 180,E1 -15349.855,E2 -15349.855} C_VEL
LIN {X 0,Y 319.428,Z 821.026,A -85,B 0,C 180,E1 -15351.973,E2 -15351.973} C_VEL
LIN {X 0,Y 320.379,Z 813.277,A -85,B 0,C 180,E1 -15353.992,E2 -15353.992} C_VEL
LIN {X 0,Y 321.496,Z 804.733,A -85,B 0,C 180,E1 -15355.776,E2 -15355.776} C_VEL
LIN {X 0,Y 322.579,Z 796.015,A -85,B 0,C 180,E1 -15357.254,E2 -15357.254} C_VEL
LIN {X 0,Y 323.89,Z 784.928,A -85,B 0,C 180,E1 -15358.774,E2 -15358.774} C_VEL
LIN {X 0,Y 325.063,Z 773.86,A -85,B 0,C 180,E1 -15359.985,E2 -15359.985} C_VEL
LIN {X 0,Y 326.215,Z 761.749,A -85,B 0,C 180,E1 -15361.005,E2 -15361.005} C_VEL
LIN {X 0,Y 324.438,Z 748.768,A -85,B 0,C 180,E1 -15361.98,E2 -15361.98} C_VEL
LIN {X 0,Y 322.062,Z 735.536,A -85,B 0,C 180,E1 -15362.726,E2 -15362.726} C_VEL
LIN {X 0,Y 320.959,Z 729.669,A -85,B 0,C 180,E1 -15362.994,E2 -15362.994} C_VEL
LIN {X 0,Y 321.738,Z 718.473,A -85,B 0,C 180,E1 -15366.848,E2 -15366.848} C_VEL
LIN {X 0,Y 322.445,Z 708.473,A -85,B 0,C 180,E1 -15370.287,E2 -15370.287} C_VEL
LIN {X 0,Y 323.062,Z 698.978,A -85,B 0,C 180,E1 -15373.573,E2 -15373.573} C_VEL
LIN {X 0,Y 323.718,Z 689.595,A -85,B 0,C 180,E1 -15376.824,E2 -15376.824} C_VEL
LIN {X 0,Y 323.964,Z 684.119,A -85,B 0,C 180,E1 -15378.742,E2 -15378.742} C_VEL
LIN {X 0,Y 323.146,Z 677.34,A -85,B 0,C 180,E1 -15381.244,E2 -15381.244} C_VEL
LIN {X 0,Y 321.997,Z 670.757,A -85,B 0,C 180,E1 -15383.735,E2 -15383.735} C_VEL
LIN {X 0,Y 320.007,Z 660.627,A -85,B 0,C 180,E1 -15387.719,E2 -15387.719} C_VEL
LIN {X 0,Y 320.152,Z 660.607,A -85,B 0,C 180,E1 -15390.001,E2 -15390.001} C_VEL
LIN {X 0,Y 320.01,Z 660.625,A -85,B 0,C 180,E1 -15392.518,E2 -15392.518} C_VEL
LIN {X 0,Y 319.947,Z 660.627,A -85,B 0,C 180,E1 -15396.306,E2 -15396.306} C_VEL
LIN {X 0,Y 319.844,Z 660.643,A -85,B 0,C 180,E1 -15398.849,E2 -15398.849} C_VEL
LIN {X 0,Y 319.687,Z 660.664,A -85,B 0,C 180,E1 -15402.7,E2 -15402.7} C_VEL
LIN {X 0,Y 319.701,Z 660.664,A -85,B 0,C 180,E1 -15405.296,E2 -15405.296} C_VEL
LIN {X 0,Y 319.691,Z 660.72,A -85,B 0,C 180,E1 -15407.018,E2 -15407.018} C_VEL
LIN {X 0,Y 323.54,Z 672.841,A -85,B 0,C 180,E1 -15408.196,E2 -15408.196} C_VEL
LIN {X 0,Y 326.629,Z 683.871,A -85,B 0,C 180,E1 -15409.482,E2 -15409.482} C_VEL
LIN {X 0,Y 326.883,Z 685.01,A -85,B 0,C 180,E1 -15409.63,E2 -15409.63} C_VEL
LIN {X 0,Y 325.859,Z 696.429,A -85,B 0,C 180,E1 -15411.012,E2 -15411.012} C_VEL
LIN {X 0,Y 324.891,Z 705.895,A -85,B 0,C 180,E1 -15412.433,E2 -15412.433} C_VEL
LIN {X 0,Y 323.723,Z 715.607,A -85,B 0,C 180,E1 -15414.243,E2 -15414.243} C_VEL
LIN {X 0,Y 322.592,Z 724.145,A -85,B 0,C 180,E1 -15416.226,E2 -15416.226} C_VEL
LIN {X 0,Y 321.657,Z 731.337,A -85,B 0,C 180,E1 -15418.374,E2 -15418.374} C_VEL
LIN {X 0,Y 321.027,Z 736.227,A -85,B 0,C 180,E1 -15420.234,E2 -15420.234} C_VEL
LIN {X 0,Y 320.441,Z 740.752,A -85,B 0,C 180,E1 -15422.503,E2 -15422.503} C_VEL
LIN {X 0,Y 320.017,Z 743.859,A -85,B 0,C 180,E1 -15424.82,E2 -15424.82} C_VEL
LIN {X 0,Y 319.877,Z 745.189,A -85,B 0,C 180,E1 -15426.386,E2 -15426.386} C_VEL
LIN {X 0,Y 319.888,Z 745.881,A -85,B 0,C 180,E1 -15427.964,E2 -15427.964} C_VEL
LIN {X 0,Y 320.062,Z 745.938,A -85,B 0,C 180,E1 -15429.777,E2 -15429.777} C_VEL
LIN {X 0,Y 320.359,Z 745.067,A -85,B 0,C 180,E1 -15431.765,E2 -15431.765} C_VEL
LIN {X 0,Y 320.826,Z 743.254,A -85,B 0,C 180,E1 -15433.706,E2 -15433.706} C_VEL
LIN {X 0,Y 321.695,Z 739.538,A -85,B 0,C 180,E1 -15436.133,E2 -15436.133} C_VEL
LIN {X 0,Y 322.452,Z 735.943,A -85,B 0,C 180,E1 -15437.821,E2 -15437.821} C_VEL
LIN {X 0,Y 323.568,Z 730.197,A -85,B 0,C 180,E1 -15439.913,E2 -15439.913} C_VEL
LIN {X 0,Y 324.704,Z 723.992,A -85,B 0,C 180,E1 -15441.685,E2 -15441.685} C_VEL
LIN {X 0,Y 325.739,Z 718.164,A -85,B 0,C 180,E1 -15443.045,E2 -15443.045} C_VEL
LIN {X 0,Y 325.722,Z 714.517,A -85,B 0,C 180,E1 -15443.861,E2 -15443.861} C_VEL
LIN {X 0,Y 324.007,Z 708.442,A -85,B 0,C 180,E1 -15445.216,E2 -15445.216} C_VEL
LIN {X 0,Y 322.378,Z 701.882,A -85,B 0,C 180,E1 -15446.499,E2 -15446.499} C_VEL
LIN {X 0,Y 322.448,Z 697.377,A -85,B 0,C 180,E1 -15447.177,E2 -15447.177} C_VEL
LIN {X 0,Y 323.09,Z 691.845,A -85,B 0,C 180,E1 -15447.87,E2 -15447.87} C_VEL
LIN {X 0,Y 320.689,Z 682.667,A -85,B 0,C 180,E1 -15449.185,E2 -15449.185} C_VEL
LIN {X 0,Y 316.752,Z 671.846,A -85,B 0,C 180,E1 -15450.6,E2 -15450.6} C_VEL
LIN {X 0,Y 312.642,Z 661.964,A -85,B 0,C 180,E1 -15451.752,E2 -15451.752} C_VEL
LIN {X 0,Y 312.587,Z 661.551,A -85,B 0,C 180,E1 -15451.826,E2 -15451.826} C_VEL
LIN {X 0,Y 312.586,Z 661.547,A -85,B 0,C 180,E1 -15454.711,E2 -15454.711} C_VEL
LIN {X 0,Y 312.541,Z 661.556,A -85,B 0,C 180,E1 -15458.913,E2 -15458.913} C_VEL
LIN {X 0,Y 312.64,Z 661.547,A -85,B 0,C 180,E1 -15461.657,E2 -15461.657} C_VEL
LIN {X 0,Y 312.696,Z 661.533,A -85,B 0,C 180,E1 -15465.686,E2 -15465.686} C_VEL
LIN {X 0,Y 312.704,Z 661.53,A -85,B 0,C 180,E1 -15469.642,E2 -15469.642} C_VEL
LIN {X 0,Y 312.874,Z 661.503,A -85,B 0,C 180,E1 -15472.254,E2 -15472.254} C_VEL
LIN {X 0,Y 312.72,Z 661.529,A -85,B 0,C 180,E1 -15474.843,E2 -15474.843} C_VEL
LIN {X 0,Y 312.993,Z 661.496,A -85,B 0,C 180,E1 -15478.714,E2 -15478.714} C_VEL
LIN {X 0,Y 312.993,Z 661.486,A -85,B 0,C 180,E1 -15481.287,E2 -15481.287} C_VEL
LIN {X 0,Y 312.72,Z 661.519,A -85,B 0,C 180,E1 -15485.158,E2 -15485.158} C_VEL
LIN {X 0,Y 312.874,Z 661.512,A -85,B 0,C 180,E1 -15487.746,E2 -15487.746} C_VEL
LIN {X 0,Y 312.671,Z 661.538,A -85,B 0,C 180,E1 -15491.671,E2 -15491.671} C_VEL
LIN {X 0,Y 312.702,Z 661.533,A -85,B 0,C 180,E1 -15494.888,E2 -15494.888} C_VEL
LIN {X 0,Y 312.633,Z 661.538,A -85,B 0,C 180,E1 -15499.237,E2 -15499.237} C_VEL
LIN {X 0,Y 312.548,Z 661.547,A -85,B 0,C 180,E1 -15502.789,E2 -15502.789} C_VEL
LIN {X 0,Y 312.599,Z 661.542,A -85,B 0,C 180,E1 -15505.933,E2 -15505.933} C_VEL
LIN {X 0,Y 312.54,Z 661.554,A -85,B 0,C 180,E1 -15509.651,E2 -15509.651} C_VEL
LIN {X 0,Y 312.522,Z 661.559,A -85,B 0,C 180,E1 -15513.689,E2 -15513.689} C_VEL
LIN {X 0,Y 312.523,Z 661.561,A -85,B 0,C 180,E1 -15517.386,E2 -15517.386} C_VEL
LIN {X 0,Y 312.509,Z 661.716,A -85,B 0,C 180,E1 -15519.182,E2 -15519.182} C_VEL
LIN {X 0,Y 313.965,Z 668.318,A -85,B 0,C 180,E1 -15523.057,E2 -15523.057} C_VEL
LIN {X 0,Y 315.354,Z 675.237,A -85,B 0,C 180,E1 -15526.695,E2 -15526.695} C_VEL
LIN {X 0,Y 316.809,Z 683.219,A -85,B 0,C 180,E1 -15530.497,E2 -15530.497} C_VEL
LIN {X 0,Y 317.122,Z 685.756,A -85,B 0,C 180,E1 -15531.645,E2 -15531.645} C_VEL
LIN {X 0,Y 316.384,Z 691.362,A -85,B 0,C 180,E1 -15533.938,E2 -15533.938} C_VEL
LIN {X 0,Y 314.896,Z 701.748,A -85,B 0,C 180,E1 -15538.006,E2 -15538.006} C_VEL
LIN {X 0,Y 313.702,Z 712.078,A -85,B 0,C 180,E1 -15541.935,E2 -15541.935} C_VEL
LIN {X 0,Y 312.737,Z 721.812,A -85,B 0,C 180,E1 -15545.527,E2 -15545.527} C_VEL
LIN {X 0,Y 315.626,Z 738.173,A -85,B 0,C 180,E1 -15546.508,E2 -15546.508} C_VEL
LIN {X 0,Y 317.002,Z 751.495,A -85,B 0,C 180,E1 -15547.496,E2 -15547.496} C_VEL
LIN {X 0,Y 317.427,Z 764.719,A -85,B 0,C 180,E1 -15548.685,E2 -15548.685} C_VEL
LIN {X 0,Y 317.449,Z 767.949,A -85,B 0,C 180,E1 -15548.97,E2 -15548.97} C_VEL
LIN {X 0,Y 317.767,Z 780.727,A -85,B 0,C 180,E1 -15549.867,E2 -15549.867} C_VEL
LIN {X 0,Y 317.751,Z 789.262,A -85,B 0,C 180,E1 -15550.623,E2 -15550.623} C_VEL
LIN {X 0,Y 316.363,Z 801.283,A -85,B 0,C 180,E1 -15551.879,E2 -15551.879} C_VEL
LIN {X 0,Y 315.104,Z 812.611,A -85,B 0,C 180,E1 -15553.417,E2 -15553.417} C_VEL
LIN {X 0,Y 313.916,Z 822.425,A -85,B 0,C 180,E1 -15555.08,E2 -15555.08} C_VEL
LIN {X 0,Y 312.738,Z 831.489,A -85,B 0,C 180,E1 -15557.013,E2 -15557.013} C_VEL
LIN {X 0,Y 311.917,Z 838.78,A -85,B 0,C 180,E1 -15558.958,E2 -15558.958} C_VEL
LIN {X 0,Y 311.358,Z 844.579,A -85,B 0,C 180,E1 -15560.908,E2 -15560.908} C_VEL
LIN {X 0,Y 311.013,Z 849.099,A -85,B 0,C 180,E1 -15562.86,E2 -15562.86} C_VEL
LIN {X 0,Y 310.836,Z 852.495,A -85,B 0,C 180,E1 -15564.81,E2 -15564.81} C_VEL
LIN {X 0,Y 310.81,Z 854.167,A -85,B 0,C 180,E1 -15566.11,E2 -15566.11} C_VEL
LIN {X 0,Y 310.766,Z 855.42,A -85,B 0,C 180,E1 -15567.407,E2 -15567.407} C_VEL
LIN {X 0,Y 310.772,Z 856.256,A -85,B 0,C 180,E1 -15568.703,E2 -15568.703} C_VEL
LIN {X 0,Y 310.818,Z 856.638,A -85,B 0,C 180,E1 -15569.999,E2 -15569.999} C_VEL
LIN {X 0,Y 310.757,Z 856.617,A -85,B 0,C 180,E1 -15571.295,E2 -15571.295} C_VEL
LIN {X 0,Y 310.761,Z 856.199,A -85,B 0,C 180,E1 -15572.592,E2 -15572.592} C_VEL
LIN {X 0,Y 310.799,Z 855.355,A -85,B 0,C 180,E1 -15573.889,E2 -15573.889} C_VEL
LIN {X 0,Y 310.84,Z 853.317,A -85,B 0,C 180,E1 -15575.827,E2 -15575.827} C_VEL
LIN {X 0,Y 311.096,Z 850.262,A -85,B 0,C 180,E1 -15577.789,E2 -15577.789} C_VEL
LIN {X 0,Y 311.619,Z 846.163,A -85,B 0,C 180,E1 -15579.738,E2 -15579.738} C_VEL
LIN {X 0,Y 312.454,Z 839.884,A -85,B 0,C 180,E1 -15582.008,E2 -15582.008} C_VEL
LIN {X 0,Y 313.608,Z 833.073,A -85,B 0,C 180,E1 -15583.939,E2 -15583.939} C_VEL
LIN {X 0,Y 314.961,Z 824.944,A -85,B 0,C 180,E1 -15585.796,E2 -15585.796} C_VEL
LIN {X 0,Y 316.385,Z 815.972,A -85,B 0,C 180,E1 -15587.449,E2 -15587.449} C_VEL
LIN {X 0,Y 318.014,Z 805.39,A -85,B 0,C 180,E1 -15589.023,E2 -15589.023} C_VEL
LIN {X 0,Y 319.654,Z 794.9,A -85,B 0,C 180,E1 -15590.259,E2 -15590.259} C_VEL
LIN {X 0,Y 320.361,Z 786.994,A -85,B 0,C 180,E1 -15591.052,E2 -15591.052} C_VEL
LIN {X 0,Y 320.486,Z 774.62,A -85,B 0,C 180,E1 -15592.131,E2 -15592.131} C_VEL
LIN {X 0,Y 320.038,Z 760.917,A -85,B 0,C 180,E1 -15593.05,E2 -15593.05} C_VEL
LIN {X 0,Y 318.298,Z 748.588,A -85,B 0,C 180,E1 -15593.748,E2 -15593.748} C_VEL
LIN {X 0,Y 315.968,Z 737.511,A -85,B 0,C 180,E1 -15594.385,E2 -15594.385} C_VEL
LIN {X 0,Y 314.654,Z 723.363,A -85,B 0,C 180,E1 -15596.243,E2 -15596.243} C_VEL
LIN {X 0,Y 313.652,Z 713.162,A -85,B 0,C 180,E1 -15597.769,E2 -15597.769} C_VEL
LIN {X 0,Y 314.982,Z 701.844,A -85,B 0,C 180,E1 -15602.019,E2 -15602.019} C_VEL
LIN {X 0,Y 316.472,Z 691.282,A -85,B 0,C 180,E1 -15606.049,E2 -15606.049} C_VEL
LIN {X 0,Y 317.052,Z 687.282,A -85,B 0,C 180,E1 -15607.609,E2 -15607.609} C_VEL
LIN {X 0,Y 316.911,Z 683.674,A -85,B 0,C 180,E1 -15609.087,E2 -15609.087} C_VEL
LIN {X 0,Y 315.314,Z 675.463,A -85,B 0,C 180,E1 -15612.647,E2 -15612.647} C_VEL
LIN {X 0,Y 313.83,Z 668.079,A -85,B 0,C 180,E1 -15616.034,E2 -15616.034} C_VEL
LIN {X 0,Y 312.56,Z 661.552,A -85,B 0,C 180,E1 -15619.195,E2 -15619.195} C_VEL
LIN {X 0,Y 312.538,Z 661.547,A -85,B 0,C 180,E1 -15622.616,E2 -15622.616} C_VEL
LIN {X 0,Y 312.516,Z 661.553,A -85,B 0,C 180,E1 -15626.31,E2 -15626.31} C_VEL
LIN {X 0,Y 312.541,Z 661.552,A -85,B 0,C 180,E1 -15630.349,E2 -15630.349} C_VEL
LIN {X 0,Y 312.599,Z 661.539,A -85,B 0,C 180,E1 -15634.064,E2 -15634.064} C_VEL
LIN {X 0,Y 312.583,Z 661.543,A -85,B 0,C 180,E1 -15637.528,E2 -15637.528} C_VEL
LIN {X 0,Y 312.634,Z 661.541,A -85,B 0,C 180,E1 -15641.656,E2 -15641.656} C_VEL
LIN {X 0,Y 312.689,Z 661.535,A -85,B 0,C 180,E1 -15645.686,E2 -15645.686} C_VEL
LIN {X 0,Y 312.704,Z 661.566,A -85,B 0,C 180,E1 -15649.314,E2 -15649.314} C_VEL
LIN {X 0,Y 315.05,Z 668.616,A -85,B 0,C 180,E1 -15652.952,E2 -15652.952} C_VEL
LIN {X 0,Y 317.582,Z 678.468,A -85,B 0,C 180,E1 -15657.463,E2 -15657.463} C_VEL
LIN {X 0,Y 318.694,Z 684.462,A -85,B 0,C 180,E1 -15660,E2 -15660} C_VEL
LIN {X 0,Y 319.167,Z 689.176,A -85,B 0,C 180,E1 -15661.893,E2 -15661.893} C_VEL
LIN {X 0,Y 318.977,Z 694.354,A -85,B 0,C 180,E1 -15663.79,E2 -15663.79} C_VEL
LIN {X 0,Y 318.063,Z 703.36,A -85,B 0,C 180,E1 -15666.98,E2 -15666.98} C_VEL
LIN {X 0,Y 317.048,Z 714.314,A -85,B 0,C 180,E1 -15670.86,E2 -15670.86} C_VEL
LIN {X 0,Y 315.968,Z 725.556,A -85,B 0,C 180,E1 -15674.82,E2 -15674.82} C_VEL
LIN {X 0,Y 315.535,Z 730.766,A -85,B 0,C 180,E1 -15676.665,E2 -15676.665} C_VEL
LIN {X 0,Y 319.332,Z 744.897,A -85,B 0,C 180,E1 -15677.656,E2 -15677.656} C_VEL
LIN {X 0,Y 321.422,Z 756.299,A -85,B 0,C 180,E1 -15678.587,E2 -15678.587} C_VEL
LIN {X 0,Y 322.253,Z 765.937,A -85,B 0,C 180,E1 -15679.459,E2 -15679.459} C_VEL
LIN {X 0,Y 320.859,Z 777.273,A -85,B 0,C 180,E1 -15680.515,E2 -15680.515} C_VEL
LIN {X 0,Y 319.26,Z 788.275,A -85,B 0,C 180,E1 -15681.807,E2 -15681.807} C_VEL
LIN {X 0,Y 317.623,Z 798.478,A -85,B 0,C 180,E1 -15683.307,E2 -15683.307} C_VEL
LIN {X 0,Y 316.036,Z 807.687,A -85,B 0,C 180,E1 -15684.994,E2 -15684.994} C_VEL
LIN {X 0,Y 314.512,Z 816.308,A -85,B 0,C 180,E1 -15686.96,E2 -15686.96} C_VEL
LIN {X 0,Y 313.239,Z 823.206,A -85,B 0,C 180,E1 -15688.954,E2 -15688.954} C_VEL
LIN {X 0,Y 312.259,Z 829.288,A -85,B 0,C 180,E1 -15691.213,E2 -15691.213} C_VEL
LIN {X 0,Y 311.482,Z 833.689,A -85,B 0,C 180,E1 -15693.403,E2 -15693.403} C_VEL
LIN {X 0,Y 310.913,Z 836.705,A -85,B 0,C 180,E1 -15695.537,E2 -15695.537} C_VEL
LIN {X 0,Y 310.62,Z 838.566,A -85,B 0,C 180,E1 -15697.654,E2 -15697.654} C_VEL
LIN {X 0,Y 310.417,Z 839.337,A -85,B 0,C 180,E1 -15699.668,E2 -15699.668} C_VEL
LIN {X 0,Y 310.361,Z 839.148,A -85,B 0,C 180,E1 -15701.647,E2 -15701.647} C_VEL
LIN {X 0,Y 310.407,Z 838.063,A -85,B 0,C 180,E1 -15703.573,E2 -15703.573} C_VEL
LIN {X 0,Y 310.637,Z 836.109,A -85,B 0,C 180,E1 -15705.465,E2 -15705.465} C_VEL
LIN {X 0,Y 310.973,Z 833.298,A -85,B 0,C 180,E1 -15707.314,E2 -15707.314} C_VEL
LIN {X 0,Y 311.475,Z 828.398,A -85,B 0,C 180,E1 -15709.634,E2 -15709.634} C_VEL
LIN {X 0,Y 312.332,Z 821.812,A -85,B 0,C 180,E1 -15711.958,E2 -15711.958} C_VEL
LIN {X 0,Y 313.202,Z 814.787,A -85,B 0,C 180,E1 -15713.882,E2 -15713.882} C_VEL
LIN {X 0,Y 314.384,Z 806.014,A -85,B 0,C 180,E1 -15715.805,E2 -15715.805} C_VEL
LIN {X 0,Y 315.661,Z 796.31,A -85,B 0,C 180,E1 -15717.513,E2 -15717.513} C_VEL
LIN {X 0,Y 316.921,Z 786.038,A -85,B 0,C 180,E1 -15718.964,E2 -15718.964} C_VEL
LIN {X 0,Y 318.209,Z 774.277,A -85,B 0,C 180,E1 -15720.295,E2 -15720.295} C_VEL
LIN {X 0,Y 319.327,Z 762.262,A -85,B 0,C 180,E1 -15721.338,E2 -15721.338} C_VEL
LIN {X 0,Y 317.589,Z 749.814,A -85,B 0,C 180,E1 -15722.309,E2 -15722.309} C_VEL
LIN {X 0,Y 315.43,Z 737.093,A -85,B 0,C 180,E1 -15723.067,E2 -15723.067} C_VEL
LIN {X 0,Y 314.044,Z 729.795,A -85,B 0,C 180,E1 -15723.412,E2 -15723.412} C_VEL
LIN {X 0,Y 314.799,Z 719.437,A -85,B 0,C 180,E1 -15727.028,E2 -15727.028} C_VEL
LIN {X 0,Y 315.51,Z 709.545,A -85,B 0,C 180,E1 -15730.481,E2 -15730.481} C_VEL
LIN {X 0,Y 316.167,Z 699.886,A -85,B 0,C 180,E1 -15733.868,E2 -15733.868} C_VEL
LIN {X 0,Y 316.902,Z 689.929,A -85,B 0,C 180,E1 -15737.368,E2 -15737.368} C_VEL
LIN {X 0,Y 317.044,Z 684.966,A -85,B 0,C 180,E1 -15739.14,E2 -15739.14} C_VEL
LIN {X 0,Y 316.167,Z 678.165,A -85,B 0,C 180,E1 -15741.693,E2 -15741.693} C_VEL
LIN {X 0,Y 314.952,Z 671.579,A -85,B 0,C 180,E1 -15744.238,E2 -15744.238} C_VEL
LIN {X 0,Y 312.958,Z 661.506,A -85,B 0,C 180,E1 -15748.231,E2 -15748.231} C_VEL
LIN {X 0,Y 313.104,Z 661.485,A -85,B 0,C 180,E1 -15750.001,E2 -15750.001} C_VEL
LIN {X 0,Y 312.953,Z 661.504,A -85,B 0,C 180,E1 -15752.575,E2 -15752.575} C_VEL
LIN {X 0,Y 312.905,Z 661.504,A -85,B 0,C 180,E1 -15756.449,E2 -15756.449} C_VEL
LIN {X 0,Y 312.789,Z 661.521,A -85,B 0,C 180,E1 -15759.05,E2 -15759.05} C_VEL
LIN {X 0,Y 312.639,Z 661.543,A -85,B 0,C 180,E1 -15762.991,E2 -15762.991} C_VEL
LIN {X 0,Y 312.656,Z 661.543,A -85,B 0,C 180,E1 -15766.571,E2 -15766.571} C_VEL
LIN {X 0,Y 316.891,Z 674.909,A -85,B 0,C 180,E1 -15767.922,E2 -15767.922} C_VEL
LIN {X 0,Y 319.872,Z 685.72,A -85,B 0,C 180,E1 -15769.243,E2 -15769.243} C_VEL
LIN {X 0,Y 319.929,Z 688.494,A -85,B 0,C 180,E1 -15769.573,E2 -15769.573} C_VEL
LIN {X 0,Y 318.845,Z 699.435,A -85,B 0,C 180,E1 -15770.989,E2 -15770.989} C_VEL
LIN {X 0,Y 317.704,Z 709.451,A -85,B 0,C 180,E1 -15772.604,E2 -15772.604} C_VEL
LIN {X 0,Y 316.566,Z 718.745,A -85,B 0,C 180,E1 -15774.463,E2 -15774.463} C_VEL
LIN {X 0,Y 315.419,Z 726.713,A -85,B 0,C 180,E1 -15776.464,E2 -15776.464} C_VEL
LIN {X 0,Y 314.506,Z 733.519,A -85,B 0,C 180,E1 -15778.628,E2 -15778.628} C_VEL
LIN {X 0,Y 313.805,Z 739.133,A -85,B 0,C 180,E1 -15781.005,E2 -15781.005} C_VEL
LIN {X 0,Y 313.388,Z 741.974,A -85,B 0,C 180,E1 -15782.563,E2 -15782.563} C_VEL
LIN {X 0,Y 313.091,Z 744.138,A -85,B 0,C 180,E1 -15784.138,E2 -15784.138} C_VEL
LIN {X 0,Y 312.866,Z 745.949,A -85,B 0,C 180,E1 -15786.033,E2 -15786.033} C_VEL
LIN {X 0,Y 312.87,Z 746.95,A -85,B 0,C 180,E1 -15788.168,E2 -15788.168} C_VEL
LIN {X 0,Y 313.174,Z 746.791,A -85,B 0,C 180,E1 -15790.602,E2 -15790.602} C_VEL
LIN {X 0,Y 313.464,Z 745.84,A -85,B 0,C 180,E1 -15792.279,E2 -15792.279} C_VEL
LIN {X 0,Y 313.992,Z 743.862,A -85,B 0,C 180,E1 -15794.255,E2 -15794.255} C_VEL
LIN {X 0,Y 314.716,Z 740.937,A -85,B 0,C 180,E1 -15796.19,E2 -15796.19} C_VEL
LIN {X 0,Y 315.809,Z 736.02,A -85,B 0,C 180,E1 -15798.525,E2 -15798.525} C_VEL
LIN {X 0,Y 316.857,Z 731.03,A -85,B 0,C 180,E1 -15800.316,E2 -15800.316} C_VEL
LIN {X 0,Y 318.237,Z 723.82,A -85,B 0,C 180,E1 -15802.357,E2 -15802.357} C_VEL
LIN {X 0,Y 319.554,Z 716.414,A -85,B 0,C 180,E1 -15804.036,E2 -15804.036} C_VEL
LIN {X 0,Y 320.851,Z 708.409,A -85,B 0,C 180,E1 -15805.524,E2 -15805.524} C_VEL
LIN {X 0,Y 322.189,Z 699.053,A -85,B 0,C 180,E1 -15806.953,E2 -15806.953} C_VEL
LIN {X 0,Y 322.448,Z 697.377,A -85,B 0,C 180,E1 -15807.177,E2 -15807.177} C_VEL
LIN {X 0,Y 322.23,Z 694.944,A -85,B 0,C 180,E1 -15807.553,E2 -15807.553} C_VEL
LIN {X 0,Y 320.509,Z 692.064,A -85,B 0,C 180,E1 -15808.121,E2 -15808.121} C_VEL
LIN {X 0,Y 315.45,Z 686.831,A -85,B 0,C 180,E1 -15809.267,E2 -15809.267} C_VEL
LIN {X 0,Y 313.947,Z 683.974,A -85,B 0,C 180,E1 -15809.735,E2 -15809.735} C_VEL
LIN {X 0,Y 309.715,Z 672.249,A -85,B 0,C 180,E1 -15811.325,E2 -15811.325} C_VEL
LIN {X 0,Y 305.584,Z 662.913,A -85,B 0,C 180,E1 -15812.476,E2 -15812.476} C_VEL
LIN {X 0,Y 305.496,Z 662.431,A -85,B 0,C 180,E1 -15812.56,E2 -15812.56} C_VEL
LIN {X 0,Y 305.507,Z 662.431,A -85,B 0,C 180,E1 -15815.539,E2 -15815.539} C_VEL
LIN {X 0,Y 305.515,Z 662.432,A -85,B 0,C 180,E1 -15819.815,E2 -15819.815} C_VEL
LIN {X 0,Y 305.576,Z 662.421,A -85,B 0,C 180,E1 -15822.603,E2 -15822.603} C_VEL
LIN {X 0,Y 305.651,Z 662.411,A -85,B 0,C 180,E1 -15825.349,E2 -15825.349} C_VEL
LIN {X 0,Y 305.64,Z 662.408,A -85,B 0,C 180,E1 -15829.4,E2 -15829.4} C_VEL
LIN {X 0,Y 305.814,Z 662.382,A -85,B 0,C 180,E1 -15832.075,E2 -15832.075} C_VEL
LIN {X 0,Y 305.691,Z 662.405,A -85,B 0,C 180,E1 -15834.724,E2 -15834.724} C_VEL
LIN {X 0,Y 305.959,Z 662.372,A -85,B 0,C 180,E1 -15838.684,E2 -15838.684} C_VEL
LIN {X 0,Y 305.959,Z 662.362,A -85,B 0,C 180,E1 -15841.316,E2 -15841.316} C_VEL
LIN {X 0,Y 305.855,Z 662.387,A -85,B 0,C 180,E1 -15846.598,E2 -15846.598} C_VEL
LIN {X 0,Y 305.738,Z 662.391,A -85,B 0,C 180,E1 -15849.26,E2 -15849.26} C_VEL
LIN {X 0,Y 305.59,Z 662.411,A -85,B 0,C 180,E1 -15853.296,E2 -15853.296} C_VEL
LIN {X 0,Y 305.596,Z 662.414,A -85,B 0,C 180,E1 -15856.02,E2 -15856.02} C_VEL
LIN {X 0,Y 305.579,Z 662.416,A -85,B 0,C 180,E1 -15859.445,E2 -15859.445} C_VEL
LIN {X 0,Y 305.493,Z 662.426,A -85,B 0,C 180,E1 -15863.041,E2 -15863.041} C_VEL
LIN {X 0,Y 305.528,Z 662.424,A -85,B 0,C 180,E1 -15866.219,E2 -15866.219} C_VEL
LIN {X 0,Y 305.491,Z 662.432,A -85,B 0,C 180,E1 -15869.047,E2 -15869.047} C_VEL
LIN {X 0,Y 305.445,Z 662.44,A -85,B 0,C 180,E1 -15871.952,E2 -15871.952} C_VEL
LIN {X 0,Y 305.465,Z 662.437,A -85,B 0,C 180,E1 -15875.113,E2 -15875.113} C_VEL
LIN {X 0,Y 305.47,Z 662.618,A -85,B 0,C 180,E1 -15878.404,E2 -15878.404} C_VEL
LIN {X 0,Y 306.856,Z 668.913,A -85,B 0,C 180,E1 -15882.286,E2 -15882.286} C_VEL
LIN {X 0,Y 308.194,Z 675.532,A -85,B 0,C 180,E1 -15885.916,E2 -15885.916} C_VEL
LIN {X 0,Y 309.613,Z 683.107,A -85,B 0,C 180,E1 -15889.69,E2 -15889.69} C_VEL
LIN {X 0,Y 310.155,Z 686.928,A -85,B 0,C 180,E1 -15891.454,E2 -15891.454} C_VEL
LIN {X 0,Y 309.676,Z 690.925,A -85,B 0,C 180,E1 -15893.167,E2 -15893.167} C_VEL
LIN {X 0,Y 308.004,Z 701.862,A -85,B 0,C 180,E1 -15897.594,E2 -15897.594} C_VEL
LIN {X 0,Y 306.61,Z 713.095,A -85,B 0,C 180,E1 -15901.972,E2 -15901.972} C_VEL
LIN {X 0,Y 305.834,Z 720.888,A -85,B 0,C 180,E1 -15904.842,E2 -15904.842} C_VEL
LIN {X 0,Y 308.51,Z 735.313,A -85,B 0,C 180,E1 -15905.73,E2 -15905.73} C_VEL
LIN {X 0,Y 310.102,Z 748.459,A -85,B 0,C 180,E1 -15906.723,E2 -15906.723} C_VEL
LIN {X 0,Y 310.652,Z 761.356,A -85,B 0,C 180,E1 -15907.886,E2 -15907.886} C_VEL
LIN {X 0,Y 310.646,Z 769.081,A -85,B 0,C 180,E1 -15908.657,E2 -15908.657} C_VEL
LIN {X 0,Y 310.921,Z 781.542,A -85,B 0,C 180,E1 -15909.577,E2 -15909.577} C_VEL
LIN {X 0,Y 310.859,Z 789.892,A -85,B 0,C 180,E1 -15910.348,E2 -15910.348} C_VEL
LIN {X 0,Y 309.567,Z 800.382,A -85,B 0,C 180,E1 -15911.467,E2 -15911.467} C_VEL
LIN {X 0,Y 308.441,Z 810.112,A -85,B 0,C 180,E1 -15912.769,E2 -15912.769} C_VEL
LIN {X 0,Y 307.267,Z 819.998,A -85,B 0,C 180,E1 -15914.409,E2 -15914.409} C_VEL
LIN {X 0,Y 306.213,Z 828.106,A -85,B 0,C 180,E1 -15916.054,E2 -15916.054} C_VEL
LIN {X 0,Y 305.107,Z 836.033,A -85,B 0,C 180,E1 -15918.035,E2 -15918.035} C_VEL
LIN {X 0,Y 304.45,Z 842.335,A -85,B 0,C 180,E1 -15920.029,E2 -15920.029} C_VEL
LIN {X 0,Y 304.042,Z 847.318,A -85,B 0,C 180,E1 -15922.027,E2 -15922.027} C_VEL
LIN {X 0,Y 303.777,Z 851.363,A -85,B 0,C 180,E1 -15924.17,E2 -15924.17} C_VEL
LIN {X 0,Y 303.722,Z 853.873,A -85,B 0,C 180,E1 -15926.019,E2 -15926.019} C_VEL
LIN {X 0,Y 303.688,Z 855.148,A -85,B 0,C 180,E1 -15927.346,E2 -15927.346} C_VEL
LIN {X 0,Y 303.683,Z 856.015,A -85,B 0,C 180,E1 -15928.673,E2 -15928.673} C_VEL
LIN {X 0,Y 303.725,Z 856.426,A -85,B 0,C 180,E1 -15929.999,E2 -15929.999} C_VEL
LIN {X 0,Y 303.67,Z 856.424,A -85,B 0,C 180,E1 -15931.325,E2 -15931.325} C_VEL
LIN {X 0,Y 303.683,Z 856.026,A -85,B 0,C 180,E1 -15932.652,E2 -15932.652} C_VEL
LIN {X 0,Y 303.71,Z 855.217,A -85,B 0,C 180,E1 -15933.98,E2 -15933.98} C_VEL
LIN {X 0,Y 303.839,Z 852.291,A -85,B 0,C 180,E1 -15936.641,E2 -15936.641} C_VEL
LIN {X 0,Y 304.191,Z 848.961,A -85,B 0,C 180,E1 -15938.636,E2 -15938.636} C_VEL
LIN {X 0,Y 304.803,Z 844.552,A -85,B 0,C 180,E1 -15940.629,E2 -15940.629} C_VEL
LIN {X 0,Y 305.645,Z 838.944,A -85,B 0,C 180,E1 -15942.617,E2 -15942.617} C_VEL
LIN {X 0,Y 306.933,Z 831.96,A -85,B 0,C 180,E1 -15944.588,E2 -15944.588} C_VEL
LIN {X 0,Y 308.258,Z 824.15,A -85,B 0,C 180,E1 -15946.367,E2 -15946.367} C_VEL
LIN {X 0,Y 309.927,Z 814.394,A -85,B 0,C 180,E1 -15948.167,E2 -15948.167} C_VEL
LIN {X 0,Y 311.573,Z 804.741,A -85,B 0,C 180,E1 -15949.604,E2 -15949.604} C_VEL
LIN {X 0,Y 313.267,Z 794.169,A -85,B 0,C 180,E1 -15950.863,E2 -15950.863} C_VEL
LIN {X 0,Y 313.819,Z 786.278,A -85,B 0,C 180,E1 -15951.685,E2 -15951.685} C_VEL
LIN {X 0,Y 314.027,Z 774.257,A -85,B 0,C 180,E1 -15952.744,E2 -15952.744} C_VEL
LIN {X 0,Y 313.647,Z 761.529,A -85,B 0,C 180,E1 -15953.627,E2 -15953.627} C_VEL
LIN {X 0,Y 311.869,Z 749.083,A -85,B 0,C 180,E1 -15954.379,E2 -15954.379} C_VEL
LIN {X 0,Y 309.427,Z 737.588,A -85,B 0,C 180,E1 -15955.068,E2 -15955.068} C_VEL
LIN {X 0,Y 308.068,Z 721.615,A -85,B 0,C 180,E1 -15957.31,E2 -15957.31} C_VEL
LIN {X 0,Y 307,Z 710.154,A -85,B 0,C 180,E1 -15959.162,E2 -15959.162} C_VEL
LIN {X 0,Y 308.33,Z 699.779,A -85,B 0,C 180,E1 -15963.164,E2 -15963.164} C_VEL
LIN {X 0,Y 309.978,Z 688.84,A -85,B 0,C 180,E1 -15967.482,E2 -15967.482} C_VEL
LIN {X 0,Y 309.97,Z 685.198,A -85,B 0,C 180,E1 -15968.988,E2 -15968.988} C_VEL
LIN {X 0,Y 308.561,Z 677.839,A -85,B 0,C 180,E1 -15972.248,E2 -15972.248} C_VEL
LIN {X 0,Y 306.718,Z 668.603,A -85,B 0,C 180,E1 -15976.574,E2 -15976.574} C_VEL
LIN {X 0,Y 305.534,Z 662.428,A -85,B 0,C 180,E1 -15979.7,E2 -15979.7} C_VEL
LIN {X 0,Y 305.497,Z 662.431,A -85,B 0,C 180,E1 -15983.626,E2 -15983.626} C_VEL
LIN {X 0,Y 305.461,Z 662.433,A -85,B 0,C 180,E1 -15986.482,E2 -15986.482} C_VEL
LIN {X 0,Y 305.492,Z 662.425,A -85,B 0,C 180,E1 -15990.949,E2 -15990.949} C_VEL
LIN {X 0,Y 305.567,Z 662.415,A -85,B 0,C 180,E1 -15994.087,E2 -15994.087} C_VEL
LIN {X 0,Y 305.523,Z 662.429,A -85,B 0,C 180,E1 -15998.404,E2 -15998.404} C_VEL
LIN {X 0,Y 305.586,Z 662.422,A -85,B 0,C 180,E1 -16001.217,E2 -16001.217} C_VEL
LIN {X 0,Y 305.644,Z 662.41,A -85,B 0,C 180,E1 -16005.349,E2 -16005.349} C_VEL
LIN {X 0,Y 305.62,Z 662.595,A -85,B 0,C 180,E1 -16007.718,E2 -16007.718} C_VEL
LIN {X 0,Y 307.94,Z 669.228,A -85,B 0,C 180,E1 -16011.469,E2 -16011.469} C_VEL
LIN {X 0,Y 309.134,Z 673.141,A -85,B 0,C 180,E1 -16013.473,E2 -16013.473} C_VEL
LIN {X 0,Y 311.185,Z 681.541,A -85,B 0,C 180,E1 -16017.411,E2 -16017.411} C_VEL
LIN {X 0,Y 312.208,Z 687.496,A -85,B 0,C 180,E1 -16020,E2 -16020} C_VEL
LIN {X 0,Y 312.564,Z 692.201,A -85,B 0,C 180,E1 -16021.933,E2 -16021.933} C_VEL
LIN {X 0,Y 312.12,Z 699.24,A -85,B 0,C 180,E1 -16024.52,E2 -16024.52} C_VEL
LIN {X 0,Y 310.896,Z 710.112,A -85,B 0,C 180,E1 -16028.449,E2 -16028.449} C_VEL
LIN {X 0,Y 309.828,Z 720.739,A -85,B 0,C 180,E1 -16032.284,E2 -16032.284} C_VEL
LIN {X 0,Y 308.861,Z 730.987,A -85,B 0,C 180,E1 -16035.952,E2 -16035.952} C_VEL
LIN {X 0,Y 312.591,Z 744.677,A -85,B 0,C 180,E1 -16036.963,E2 -16036.963} C_VEL
LIN {X 0,Y 314.912,Z 756.997,A -85,B 0,C 180,E1 -16038.017,E2 -16038.017} C_VEL
LIN {X 0,Y 315.835,Z 766.542,A -85,B 0,C 180,E1 -16038.923,E2 -16038.923} C_VEL
LIN {X 0,Y 314.131,Z 779.569,A -85,B 0,C 180,E1 -16040.188,E2 -16040.188} C_VEL
LIN {X 0,Y 312.35,Z 790.924,A -85,B 0,C 180,E1 -16041.62,E2 -16041.62} C_VEL
LIN {X 0,Y 310.461,Z 801.722,A -85,B 0,C 180,E1 -16043.338,E2 -16043.338} C_VEL
LIN {X 0,Y 308.874,Z 810.403,A -85,B 0,C 180,E1 -16045.079,E2 -16045.079} C_VEL
LIN {X 0,Y 307.276,Z 818.964,A -85,B 0,C 180,E1 -16047.222,E2 -16047.222} C_VEL
LIN {X 0,Y 306.008,Z 825.299,A -85,B 0,C 180,E1 -16049.224,E2 -16049.224} C_VEL
LIN {X 0,Y 305.061,Z 830.871,A -85,B 0,C 180,E1 -16051.528,E2 -16051.528} C_VEL
LIN {X 0,Y 304.291,Z 834.865,A -85,B 0,C 180,E1 -16053.752,E2 -16053.752} C_VEL
LIN {X 0,Y 303.751,Z 837.554,A -85,B 0,C 180,E1 -16055.925,E2 -16055.925} C_VEL
LIN {X 0,Y 303.461,Z 839.099,A -85,B 0,C 180,E1 -16058.057,E2 -16058.057} C_VEL
LIN {X 0,Y 303.275,Z 839.58,A -85,B 0,C 180,E1 -16060.456,E2 -16060.456} C_VEL
LIN {X 0,Y 303.266,Z 839.102,A -85,B 0,C 180,E1 -16062.226,E2 -16062.226} C_VEL
LIN {X 0,Y 303.357,Z 837.789,A -85,B 0,C 180,E1 -16064.096,E2 -16064.096} C_VEL
LIN {X 0,Y 303.629,Z 835.578,A -85,B 0,C 180,E1 -16066.022,E2 -16066.022} C_VEL
LIN {X 0,Y 303.992,Z 832.529,A -85,B 0,C 180,E1 -16067.899,E2 -16067.899} C_VEL
LIN {X 0,Y 304.548,Z 827.535,A -85,B 0,C 180,E1 -16070.181,E2 -16070.181} C_VEL
LIN {X 0,Y 305.417,Z 820.959,A -85,B 0,C 180,E1 -16072.441,E2 -16072.441} C_VEL
LIN {X 0,Y 306.316,Z 814.165,A -85,B 0,C 180,E1 -16074.29,E2 -16074.29} C_VEL
LIN {X 0,Y 307.496,Z 805.762,A -85,B 0,C 180,E1 -16076.145,E2 -16076.145} C_VEL
LIN {X 0,Y 308.684,Z 797.081,A -85,B 0,C 180,E1 -16077.708,E2 -16077.708} C_VEL
LIN {X 0,Y 310.03,Z 786.325,A -85,B 0,C 180,E1 -16079.271,E2 -16079.271} C_VEL
LIN {X 0,Y 311.341,Z 774.888,A -85,B 0,C 180,E1 -16080.597,E2 -16080.597} C_VEL
LIN {X 0,Y 312.501,Z 763.753,A -85,B 0,C 180,E1 -16081.603,E2 -16081.603} C_VEL
LIN {X 0,Y 311.066,Z 752.368,A -85,B 0,C 180,E1 -16082.538,E2 -16082.538} C_VEL
LIN {X 0,Y 308.816,Z 738.857,A -85,B 0,C 180,E1 -16083.409,E2 -16083.409} C_VEL
LIN {X 0,Y 307.154,Z 729.929,A -85,B 0,C 180,E1 -16083.854,E2 -16083.854} C_VEL
LIN {X 0,Y 308.027,Z 718.502,A -85,B 0,C 180,E1 -16087.886,E2 -16087.886} C_VEL
LIN {X 0,Y 308.884,Z 706.57,A -85,B 0,C 180,E1 -16092.113,E2 -16092.113} C_VEL
LIN {X 0,Y 309.788,Z 695.034,A -85,B 0,C 180,E1 -16096.22,E2 -16096.22} C_VEL
LIN {X 0,Y 310.197,Z 687.581,A -85,B 0,C 180,E1 -16098.897,E2 -16098.897} C_VEL
LIN {X 0,Y 309.431,Z 680.689,A -85,B 0,C 180,E1 -16101.511,E2 -16101.511} C_VEL
LIN {X 0,Y 308.259,Z 674.035,A -85,B 0,C 180,E1 -16104.112,E2 -16104.112} C_VEL
LIN {X 0,Y 305.971,Z 662.376,A -85,B 0,C 180,E1 -16108.849,E2 -16108.849} C_VEL
LIN {X 0,Y 305.961,Z 662.372,A -85,B 0,C 180,E1 -16111.317,E2 -16111.317} C_VEL
LIN {X 0,Y 305.689,Z 662.409,A -85,B 0,C 180,E1 -16115.277,E2 -16115.277} C_VEL
LIN {X 0,Y 305.81,Z 662.394,A -85,B 0,C 180,E1 -16117.926,E2 -16117.926} C_VEL
LIN {X 0,Y 305.608,Z 662.418,A -85,B 0,C 180,E1 -16121.946,E2 -16121.946} C_VEL
LIN {X 0,Y 305.629,Z 662.417,A -85,B 0,C 180,E1 -16125.029,E2 -16125.029} C_VEL
LIN {X 0,Y 305.592,Z 662.421,A -85,B 0,C 180,E1 -16126.115,E2 -16126.115} C_VEL
LIN {X 0,Y 309.85,Z 675.501,A -85,B 0,C 180,E1 -16127.49,E2 -16127.49} C_VEL
LIN {X 0,Y 312.944,Z 686.731,A -85,B 0,C 180,E1 -16128.886,E2 -16128.886} C_VEL
LIN {X 0,Y 313.148,Z 689.56,A -85,B 0,C 180,E1 -16129.24,E2 -16129.24} C_VEL
LIN {X 0,Y 312.095,Z 699.922,A -85,B 0,C 180,E1 -16130.601,E2 -16130.601} C_VEL
LIN {X 0,Y 310.867,Z 710.242,A -85,B 0,C 180,E1 -16132.289,E2 -16132.289} C_VEL
LIN {X 0,Y 309.715,Z 719.235,A -85,B 0,C 180,E1 -16134.108,E2 -16134.108} C_VEL
LIN {X 0,Y 308.636,Z 726.768,A -85,B 0,C 180,E1 -16135.999,E2 -16135.999} C_VEL
LIN {X 0,Y 307.612,Z 734.008,A -85,B 0,C 180,E1 -16138.299,E2 -16138.299} C_VEL
LIN {X 0,Y 306.995,Z 738.766,A -85,B 0,C 180,E1 -16140.242,E2 -16140.242} C_VEL
LIN {X 0,Y 306.341,Z 743.179,A -85,B 0,C 180,E1 -16142.634,E2 -16142.634} C_VEL
LIN {X 0,Y 305.942,Z 746.144,A -85,B 0,C 180,E1 -16145.051,E2 -16145.051} C_VEL
LIN {X 0,Y 305.839,Z 747.4,A -85,B 0,C 180,E1 -16146.689,E2 -16146.689} C_VEL
LIN {X 0,Y 305.893,Z 748.075,A -85,B 0,C 180,E1 -16148.633,E2 -16148.633} C_VEL
LIN {X 0,Y 306.179,Z 747.829,A -85,B 0,C 180,E1 -16150.758,E2 -16150.758} C_VEL
LIN {X 0,Y 306.743,Z 746.059,A -85,B 0,C 180,E1 -16153.421,E2 -16153.421} C_VEL
LIN {X 0,Y 307.293,Z 744.029,A -85,B 0,C 180,E1 -16155.153,E2 -16155.153} C_VEL
LIN {X 0,Y 308.038,Z 741.209,A -85,B 0,C 180,E1 -16156.895,E2 -16156.895} C_VEL
LIN {X 0,Y 309.129,Z 736.387,A -85,B 0,C 180,E1 -16159.107,E2 -16159.107} C_VEL
LIN {X 0,Y 310.554,Z 729.909,A -85,B 0,C 180,E1 -16161.342,E2 -16161.342} C_VEL
LIN {X 0,Y 311.898,Z 723.255,A -85,B 0,C 180,E1 -16163.156,E2 -16163.156} C_VEL
LIN {X 0,Y 313.306,Z 715.328,A -85,B 0,C 180,E1 -16164.911,E2 -16164.911} C_VEL
LIN {X 0,Y 315.027,Z 705.229,A -85,B 0,C 180,E1 -16166.677,E2 -16166.677} C_VEL
LIN {X 0,Y 316.515,Z 694.733,A -85,B 0,C 180,E1 -16168.15,E2 -16168.15} C_VEL
LIN {X 0,Y 316.326,Z 692.381,A -85,B 0,C 180,E1 -16168.479,E2 -16168.479} C_VEL
LIN {X 0,Y 313.947,Z 683.974,A -85,B 0,C 180,E1 -16169.735,E2 -16169.735} C_VEL
LIN {X 0,Y 312.43,Z 681.281,A -85,B 0,C 180,E1 -16170.187,E2 -16170.187} C_VEL
LIN {X 0,Y 308.41,Z 677.991,A -85,B 0,C 180,E1 -16170.972,E2 -16170.972} C_VEL
LIN {X 0,Y 304.138,Z 674.735,A -85,B 0,C 180,E1 -16171.753,E2 -16171.753} C_VEL
LIN {X 0,Y 302.229,Z 672.062,A -85,B 0,C 180,E1 -16172.192,E2 -16172.192} C_VEL
LIN {X 0,Y 298.607,Z 664.056,A -85,B 0,C 180,E1 -16173.225,E2 -16173.225} C_VEL
LIN {X 0,Y 298.475,Z 663.299,A -85,B 0,C 180,E1 -16173.339,E2 -16173.339} C_VEL
LIN {X 0,Y 298.432,Z 663.301,A -85,B 0,C 180,E1 -16176.7,E2 -16176.7} C_VEL
LIN {X 0,Y 298.54,Z 663.299,A -85,B 0,C 180,E1 -16180.757,E2 -16180.757} C_VEL
LIN {X 0,Y 298.595,Z 663.292,A -85,B 0,C 180,E1 -16184.995,E2 -16184.995} C_VEL
LIN {X 0,Y 298.595,Z 663.285,A -85,B 0,C 180,E1 -16189.147,E2 -16189.147} C_VEL
LIN {X 0,Y 298.76,Z 663.262,A -85,B 0,C 180,E1 -16191.886,E2 -16191.886} C_VEL
LIN {X 0,Y 298.662,Z 663.282,A -85,B 0,C 180,E1 -16194.599,E2 -16194.599} C_VEL
LIN {X 0,Y 298.926,Z 663.248,A -85,B 0,C 180,E1 -16198.653,E2 -16198.653} C_VEL
LIN {X 0,Y 298.926,Z 663.238,A -85,B 0,C 180,E1 -16201.347,E2 -16201.347} C_VEL
LIN {X 0,Y 298.8,Z 663.265,A -85,B 0,C 180,E1 -16206.754,E2 -16206.754} C_VEL
LIN {X 0,Y 298.683,Z 663.27,A -85,B 0,C 180,E1 -16209.481,E2 -16209.481} C_VEL
LIN {X 0,Y 298.554,Z 663.289,A -85,B 0,C 180,E1 -16213.616,E2 -16213.616} C_VEL
LIN {X 0,Y 298.551,Z 663.289,A -85,B 0,C 180,E1 -16216.409,E2 -16216.409} C_VEL
LIN {X 0,Y 298.514,Z 663.295,A -85,B 0,C 180,E1 -16219.655,E2 -16219.655} C_VEL
LIN {X 0,Y 298.46,Z 663.303,A -85,B 0,C 180,E1 -16223.598,E2 -16223.598} C_VEL
LIN {X 0,Y 298.488,Z 663.303,A -85,B 0,C 180,E1 -16226.575,E2 -16226.575} C_VEL
LIN {X 0,Y 298.419,Z 663.314,A -85,B 0,C 180,E1 -16229.641,E2 -16229.641} C_VEL
LIN {X 0,Y 298.397,Z 663.315,A -85,B 0,C 180,E1 -16232.8,E2 -16232.8} C_VEL
LIN {X 0,Y 298.447,Z 663.311,A -85,B 0,C 180,E1 -16236.807,E2 -16236.807} C_VEL
LIN {X 0,Y 298.467,Z 663.345,A -85,B 0,C 180,E1 -16237.483,E2 -16237.483} C_VEL
LIN {X 0,Y 299.704,Z 669.375,A -85,B 0,C 180,E1 -16241.375,E2 -16241.375} C_VEL
LIN {X 0,Y 300.823,Z 674.786,A -85,B 0,C 180,E1 -16244.498,E2 -16244.498} C_VEL
LIN {X 0,Y 302.121,Z 681.606,A -85,B 0,C 180,E1 -16248.107,E2 -16248.107} C_VEL
LIN {X 0,Y 303.174,Z 688.032,A -85,B 0,C 180,E1 -16251.251,E2 -16251.251} C_VEL
LIN {X 0,Y 302.783,Z 691.737,A -85,B 0,C 180,E1 -16252.879,E2 -16252.879} C_VEL
LIN {X 0,Y 301.092,Z 702.072,A -85,B 0,C 180,E1 -16257.172,E2 -16257.172} C_VEL
LIN {X 0,Y 299.543,Z 714.15,A -85,B 0,C 180,E1 -16262.014,E2 -16262.014} C_VEL
LIN {X 0,Y 298.955,Z 719.422,A -85,B 0,C 180,E1 -16264.08,E2 -16264.08} C_VEL
LIN {X 0,Y 301.77,Z 734.456,A -85,B 0,C 180,E1 -16265.049,E2 -16265.049} C_VEL
LIN {X 0,Y 303.372,Z 747.686,A -85,B 0,C 180,E1 -16266.09,E2 -16266.09} C_VEL
LIN {X 0,Y 303.966,Z 760.327,A -85,B 0,C 180,E1 -16267.281,E2 -16267.281} C_VEL
LIN {X 0,Y 303.871,Z 770.099,A -85,B 0,C 180,E1 -16268.325,E2 -16268.325} C_VEL
LIN {X 0,Y 304.077,Z 781.302,A -85,B 0,C 180,E1 -16269.184,E2 -16269.184} C_VEL
LIN {X 0,Y 303.968,Z 790.518,A -85,B 0,C 180,E1 -16270.06,E2 -16270.06} C_VEL
LIN {X 0,Y 302.471,Z 802.099,A -85,B 0,C 180,E1 -16271.368,E2 -16271.368} C_VEL
LIN {X 0,Y 301.222,Z 812.688,A -85,B 0,C 180,E1 -16272.892,E2 -16272.892} C_VEL
LIN {X 0,Y 300.156,Z 821.111,A -85,B 0,C 180,E1 -16274.379,E2 -16274.379} C_VEL
LIN {X 0,Y 299.073,Z 829.002,A -85,B 0,C 180,E1 -16276.062,E2 -16276.062} C_VEL
LIN {X 0,Y 297.978,Z 836.667,A -85,B 0,C 180,E1 -16278.089,E2 -16278.089} C_VEL
LIN {X 0,Y 297.26,Z 843.722,A -85,B 0,C 180,E1 -16280.473,E2 -16280.473} C_VEL
LIN {X 0,Y 296.868,Z 848.363,A -85,B 0,C 180,E1 -16282.518,E2 -16282.518} C_VEL
LIN {X 0,Y 296.67,Z 851.855,A -85,B 0,C 180,E1 -16284.562,E2 -16284.562} C_VEL
LIN {X 0,Y 296.638,Z 853.579,A -85,B 0,C 180,E1 -16285.923,E2 -16285.923} C_VEL
LIN {X 0,Y 296.612,Z 854.874,A -85,B 0,C 180,E1 -16287.283,E2 -16287.283} C_VEL
LIN {X 0,Y 296.597,Z 855.762,A -85,B 0,C 180,E1 -16288.642,E2 -16288.642} C_VEL
LIN {X 0,Y 296.634,Z 856.213,A -85,B 0,C 180,E1 -16289.999,E2 -16289.999} C_VEL
LIN {X 0,Y 296.584,Z 856.232,A -85,B 0,C 180,E1 -16291.357,E2 -16291.357} C_VEL
LIN {X 0,Y 296.606,Z 855.857,A -85,B 0,C 180,E1 -16292.715,E2 -16292.715} C_VEL
LIN {X 0,Y 296.605,Z 855.083,A -85,B 0,C 180,E1 -16294.076,E2 -16294.076} C_VEL
LIN {X 0,Y 296.629,Z 853.602,A -85,B 0,C 180,E1 -16295.669,E2 -16295.669} C_VEL
LIN {X 0,Y 296.988,Z 850.156,A -85,B 0,C 180,E1 -16298.162,E2 -16298.162} C_VEL
LIN {X 0,Y 297.555,Z 846.17,A -85,B 0,C 180,E1 -16300.203,E2 -16300.203} C_VEL
LIN {X 0,Y 298.524,Z 840.037,A -85,B 0,C 180,E1 -16302.577,E2 -16302.577} C_VEL
LIN {X 0,Y 300.07,Z 832.133,A -85,B 0,C 180,E1 -16304.929,E2 -16304.929} C_VEL
LIN {X 0,Y 301.371,Z 824.938,A -85,B 0,C 180,E1 -16306.646,E2 -16306.646} C_VEL
LIN {X 0,Y 302.879,Z 816.741,A -85,B 0,C 180,E1 -16308.254,E2 -16308.254} C_VEL
LIN {X 0,Y 304.701,Z 806.444,A -85,B 0,C 180,E1 -16309.889,E2 -16309.889} C_VEL
LIN {X 0,Y 306.691,Z 794.968,A -85,B 0,C 180,E1 -16311.332,E2 -16311.332} C_VEL
LIN {X 0,Y 307.298,Z 787.208,A -85,B 0,C 180,E1 -16312.169,E2 -16312.169} C_VEL
LIN {X 0,Y 307.64,Z 774.882,A -85,B 0,C 180,E1 -16313.307,E2 -16313.307} C_VEL
LIN {X 0,Y 307.4,Z 763.056,A -85,B 0,C 180,E1 -16314.178,E2 -16314.178} C_VEL
LIN {X 0,Y 305.811,Z 751.15,A -85,B 0,C 180,E1 -16314.954,E2 -16314.954} C_VEL
LIN {X 0,Y 302.928,Z 737.463,A -85,B 0,C 180,E1 -16315.82,E2 -16315.82} C_VEL
LIN {X 0,Y 301.787,Z 723.239,A -85,B 0,C 180,E1 -16317.928,E2 -16317.928} C_VEL
LIN {X 0,Y 300.848,Z 712.392,A -85,B 0,C 180,E1 -16319.749,E2 -16319.749} C_VEL
LIN {X 0,Y 300.406,Z 706.608,A -85,B 0,C 180,E1 -16320.827,E2 -16320.827} C_VEL
LIN {X 0,Y 301.8,Z 696.786,A -85,B 0,C 180,E1 -16324.748,E2 -16324.748} C_VEL
LIN {X 0,Y 303.049,Z 688.882,A -85,B 0,C 180,E1 -16327.955,E2 -16327.955} C_VEL
LIN {X 0,Y 302.884,Z 685.655,A -85,B 0,C 180,E1 -16329.349,E2 -16329.349} C_VEL
LIN {X 0,Y 301.248,Z 677.468,A -85,B 0,C 180,E1 -16333.084,E2 -16333.084} C_VEL
LIN {X 0,Y 299.59,Z 669.095,A -85,B 0,C 180,E1 -16337.132,E2 -16337.132} C_VEL
LIN {X 0,Y 298.456,Z 663.309,A -85,B 0,C 180,E1 -16340.192,E2 -16340.192} C_VEL
LIN {X 0,Y 298.429,Z 663.313,A -85,B 0,C 180,E1 -16343.931,E2 -16343.931} C_VEL
LIN {X 0,Y 298.391,Z 663.309,A -85,B 0,C 180,E1 -16347.983,E2 -16347.983} C_VEL
LIN {X 0,Y 298.46,Z 663.301,A -85,B 0,C 180,E1 -16351.904,E2 -16351.904} C_VEL
LIN {X 0,Y 298.481,Z 663.299,A -85,B 0,C 180,E1 -16354.923,E2 -16354.923} C_VEL
LIN {X 0,Y 298.455,Z 663.304,A -85,B 0,C 180,E1 -16359.315,E2 -16359.315} C_VEL
LIN {X 0,Y 298.533,Z 663.293,A -85,B 0,C 180,E1 -16362.179,E2 -16362.179} C_VEL
LIN {X 0,Y 298.576,Z 663.303,A -85,B 0,C 180,E1 -16365.691,E2 -16365.691} C_VEL
LIN {X 0,Y 300.757,Z 669.777,A -85,B 0,C 180,E1 -16369.716,E2 -16369.716} C_VEL
LIN {X 0,Y 302.519,Z 675.055,A -85,B 0,C 180,E1 -16372.659,E2 -16372.659} C_VEL
LIN {X 0,Y 304.797,Z 684.63,A -85,B 0,C 180,E1 -16377.357,E2 -16377.357} C_VEL
LIN {X 0,Y 305.708,Z 690.498,A -85,B 0,C 180,E1 -16380,E2 -16380} C_VEL
LIN {X 0,Y 306.042,Z 695.391,A -85,B 0,C 180,E1 -16381.974,E2 -16381.974} C_VEL
LIN {X 0,Y 305.382,Z 702.318,A -85,B 0,C 180,E1 -16384.62,E2 -16384.62} C_VEL
LIN {X 0,Y 304.088,Z 713.284,A -85,B 0,C 180,E1 -16388.64,E2 -16388.64} C_VEL
LIN {X 0,Y 302.941,Z 723.906,A -85,B 0,C 180,E1 -16392.547,E2 -16392.547} C_VEL
LIN {X 0,Y 302.244,Z 731.35,A -85,B 0,C 180,E1 -16395.208,E2 -16395.208} C_VEL
LIN {X 0,Y 306.119,Z 745.16,A -85,B 0,C 180,E1 -16396.286,E2 -16396.286} C_VEL
LIN {X 0,Y 308.209,Z 755.958,A -85,B 0,C 180,E1 -16397.243,E2 -16397.243} C_VEL
LIN {X 0,Y 309.408,Z 767.473,A -85,B 0,C 180,E1 -16398.392,E2 -16398.392} C_VEL
LIN {X 0,Y 307.893,Z 778.702,A -85,B 0,C 180,E1 -16399.501,E2 -16399.501} C_VEL
LIN {X 0,Y 306.261,Z 788.937,A -85,B 0,C 180,E1 -16400.765,E2 -16400.765} C_VEL
LIN {X 0,Y 304.538,Z 798.45,A -85,B 0,C 180,E1 -16402.214,E2 -16402.214} C_VEL
LIN {X 0,Y 302.758,Z 807.711,A -85,B 0,C 180,E1 -16403.968,E2 -16403.968} C_VEL
LIN {X 0,Y 301.102,Z 816.136,A -85,B 0,C 180,E1 -16405.953,E2 -16405.953} C_VEL
LIN {X 0,Y 299.667,Z 822.986,A -85,B 0,C 180,E1 -16407.973,E2 -16407.973} C_VEL
LIN {X 0,Y 298.416,Z 829.395,A -85,B 0,C 180,E1 -16410.421,E2 -16410.421} C_VEL
LIN {X 0,Y 297.477,Z 834.211,A -85,B 0,C 180,E1 -16412.914,E2 -16412.914} C_VEL
LIN {X 0,Y 296.97,Z 836.583,A -85,B 0,C 180,E1 -16414.609,E2 -16414.609} C_VEL
LIN {X 0,Y 296.59,Z 838.296,A -85,B 0,C 180,E1 -16416.327,E2 -16416.327} C_VEL
LIN {X 0,Y 296.319,Z 839.53,A -85,B 0,C 180,E1 -16418.495,E2 -16418.495} C_VEL
LIN {X 0,Y 296.175,Z 839.749,A -85,B 0,C 180,E1 -16420.596,E2 -16420.596} C_VEL
LIN {X 0,Y 296.174,Z 839.037,A -85,B 0,C 180,E1 -16422.643,E2 -16422.643} C_VEL
LIN {X 0,Y 296.407,Z 836.689,A -85,B 0,C 180,E1 -16425.342,E2 -16425.342} C_VEL
LIN {X 0,Y 296.75,Z 834.002,A -85,B 0,C 180,E1 -16427.238,E2 -16427.238} C_VEL
LIN {X 0,Y 297.15,Z 830.309,A -85,B 0,C 180,E1 -16429.186,E2 -16429.186} C_VEL
LIN {X 0,Y 297.799,Z 825.518,A -85,B 0,C 180,E1 -16431.15,E2 -16431.15} C_VEL
LIN {X 0,Y 298.635,Z 819.417,A -85,B 0,C 180,E1 -16433.144,E2 -16433.144} C_VEL
LIN {X 0,Y 299.701,Z 811.684,A -85,B 0,C 180,E1 -16435.16,E2 -16435.16} C_VEL
LIN {X 0,Y 301.05,Z 801.95,A -85,B 0,C 180,E1 -16437.184,E2 -16437.184} C_VEL
LIN {X 0,Y 302.518,Z 791.775,A -85,B 0,C 180,E1 -16438.863,E2 -16438.863} C_VEL
LIN {X 0,Y 303.923,Z 780.298,A -85,B 0,C 180,E1 -16440.379,E2 -16440.379} C_VEL
LIN {X 0,Y 305.179,Z 769.187,A -85,B 0,C 180,E1 -16441.532,E2 -16441.532} C_VEL
LIN {X 0,Y 305.536,Z 763.249,A -85,B 0,C 180,E1 -16442.053,E2 -16442.053} C_VEL
LIN {X 0,Y 303.722,Z 749.84,A -85,B 0,C 180,E1 -16443.151,E2 -16443.151} C_VEL
LIN {X 0,Y 301.369,Z 736.407,A -85,B 0,C 180,E1 -16443.979,E2 -16443.979} C_VEL
LIN {X 0,Y 300.217,Z 730.1,A -85,B 0,C 180,E1 -16444.291,E2 -16444.291} C_VEL
LIN {X 0,Y 301.161,Z 718.109,A -85,B 0,C 180,E1 -16448.594,E2 -16448.594} C_VEL
LIN {X 0,Y 302.011,Z 707.02,A -85,B 0,C 180,E1 -16452.572,E2 -16452.572} C_VEL
LIN {X 0,Y 302.941,Z 695.895,A -85,B 0,C 180,E1 -16456.586,E2 -16456.586} C_VEL
LIN {X 0,Y 303.292,Z 690.237,A -85,B 0,C 180,E1 -16458.641,E2 -16458.641} C_VEL
LIN {X 0,Y 302.938,Z 684.943,A -85,B 0,C 180,E1 -16460.655,E2 -16460.655} C_VEL
LIN {X 0,Y 301.87,Z 678.173,A -85,B 0,C 180,E1 -16463.316,E2 -16463.316} C_VEL
LIN {X 0,Y 299.624,Z 666.649,A -85,B 0,C 180,E1 -16467.984,E2 -16467.984} C_VEL
LIN {X 0,Y 298.967,Z 663.245,A -85,B 0,C 180,E1 -16469.411,E2 -16469.411} C_VEL
LIN {X 0,Y 298.849,Z 663.261,A -85,B 0,C 180,E1 -16472.697,E2 -16472.697} C_VEL
LIN {X 0,Y 298.794,Z 663.261,A -85,B 0,C 180,E1 -16476.755,E2 -16476.755} C_VEL
LIN {X 0,Y 298.682,Z 663.275,A -85,B 0,C 180,E1 -16479.481,E2 -16479.481} C_VEL
LIN {X 0,Y 298.552,Z 663.298,A -85,B 0,C 180,E1 -16483.616,E2 -16483.616} C_VEL
LIN {X 0,Y 298.578,Z 663.294,A -85,B 0,C 180,E1 -16485.674,E2 -16485.674} C_VEL
LIN {X 0,Y 302.77,Z 676.171,A -85,B 0,C 180,E1 -16487.042,E2 -16487.042} C_VEL
LIN {X 0,Y 305.952,Z 687.626,A -85,B 0,C 180,E1 -16488.499,E2 -16488.499} C_VEL
LIN {X 0,Y 306.399,Z 690.411,A -85,B 0,C 180,E1 -16488.875,E2 -16488.875} C_VEL
LIN {X 0,Y 305.348,Z 700.361,A -85,B 0,C 180,E1 -16490.197,E2 -16490.197} C_VEL
LIN {X 0,Y 304.072,Z 710.767,A -85,B 0,C 180,E1 -16491.919,E2 -16491.919} C_VEL
LIN {X 0,Y 302.982,Z 718.987,A -85,B 0,C 180,E1 -16493.587,E2 -16493.587} C_VEL
LIN {X 0,Y 301.852,Z 726.798,A -85,B 0,C 180,E1 -16495.522,E2 -16495.522} C_VEL
LIN {X 0,Y 300.784,Z 734.215,A -85,B 0,C 180,E1 -16497.861,E2 -16497.861} C_VEL
LIN {X 0,Y 300.052,Z 739.332,A -85,B 0,C 180,E1 -16499.93,E2 -16499.93} C_VEL
LIN {X 0,Y 299.383,Z 743.801,A -85,B 0,C 180,E1 -16502.318,E2 -16502.318} C_VEL
LIN {X 0,Y 298.957,Z 746.781,A -85,B 0,C 180,E1 -16504.635,E2 -16504.635} C_VEL
LIN {X 0,Y 298.802,Z 748.512,A -85,B 0,C 180,E1 -16506.899,E2 -16506.899} C_VEL
LIN {X 0,Y 298.948,Z 749.126,A -85,B 0,C 180,E1 -16509.402,E2 -16509.402} C_VEL
LIN {X 0,Y 299.264,Z 748.705,A -85,B 0,C 180,E1 -16511.28,E2 -16511.28} C_VEL
LIN {X 0,Y 299.742,Z 747.334,A -85,B 0,C 180,E1 -16513.377,E2 -16513.377} C_VEL
LIN {X 0,Y 300.397,Z 745.039,A -85,B 0,C 180,E1 -16515.423,E2 -16515.423} C_VEL
LIN {X 0,Y 301.292,Z 741.782,A -85,B 0,C 180,E1 -16517.432,E2 -16517.432} C_VEL
LIN {X 0,Y 302.293,Z 737.593,A -85,B 0,C 180,E1 -16519.385,E2 -16519.385} C_VEL
LIN {X 0,Y 303.561,Z 732.292,A -85,B 0,C 180,E1 -16521.311,E2 -16521.311} C_VEL
LIN {X 0,Y 304.908,Z 725.88,A -85,B 0,C 180,E1 -16523.181,E2 -16523.181} C_VEL
LIN {X 0,Y 306.441,Z 718.076,A -85,B 0,C 180,E1 -16525.015,E2 -16525.015} C_VEL
LIN {X 0,Y 308.215,Z 708.466,A -85,B 0,C 180,E1 -16526.821,E2 -16526.821} C_VEL
LIN {X 0,Y 309.778,Z 698.098,A -85,B 0,C 180,E1 -16528.368,E2 -16528.368} C_VEL
LIN {X 0,Y 310.019,Z 695.205,A -85,B 0,C 180,E1 -16528.764,E2 -16528.764} C_VEL
LIN {X 0,Y 307.166,Z 685.147,A -85,B 0,C 180,E1 -16530.345,E2 -16530.345} C_VEL
LIN {X 0,Y 303.362,Z 674.667,A -85,B 0,C 180,E1 -16531.834,E2 -16531.834} C_VEL
LIN {X 0,Y 302.229,Z 672.062,A -85,B 0,C 180,E1 -16532.192,E2 -16532.192} C_VEL
LIN {X 0,Y 300.935,Z 670.669,A -85,B 0,C 180,E1 -16532.457,E2 -16532.457} C_VEL
LIN {X 0,Y 297.82,Z 669.645,A -85,B 0,C 180,E1 -16532.922,E2 -16532.922} C_VEL
LIN {X 0,Y 293.901,Z 668.512,A -85,B 0,C 180,E1 -16533.499,E2 -16533.499} C_VEL
LIN {X 0,Y 292.883,Z 667.658,A -85,B 0,C 180,E1 -16533.69,E2 -16533.69} C_VEL
LIN {X 0,Y 291.601,Z 665.031,A -85,B 0,C 180,E1 -16534.048,E2 -16534.048} C_VEL
LIN {X 0,Y 291.419,Z 664.178,A -85,B 0,C 180,E1 -16534.151,E2 -16534.151} C_VEL
LIN {X 0,Y 291.376,Z 664.179,A -85,B 0,C 180,E1 -16537.299,E2 -16537.299} C_VEL
LIN {X 0,Y 291.46,Z 664.18,A -85,B 0,C 180,E1 -16540.27,E2 -16540.27} C_VEL
LIN {X 0,Y 291.557,Z 664.17,A -85,B 0,C 180,E1 -16544.624,E2 -16544.624} C_VEL
LIN {X 0,Y 291.539,Z 664.163,A -85,B 0,C 180,E1 -16548.881,E2 -16548.881} C_VEL
LIN {X 0,Y 291.711,Z 664.141,A -85,B 0,C 180,E1 -16551.689,E2 -16551.689} C_VEL
LIN {X 0,Y 291.633,Z 664.158,A -85,B 0,C 180,E1 -16554.469,E2 -16554.469} C_VEL
LIN {X 0,Y 291.892,Z 664.125,A -85,B 0,C 180,E1 -16558.621,E2 -16558.621} C_VEL
LIN {X 0,Y 291.892,Z 664.114,A -85,B 0,C 180,E1 -16561.38,E2 -16561.38} C_VEL
LIN {X 0,Y 291.749,Z 664.143,A -85,B 0,C 180,E1 -16566.918,E2 -16566.918} C_VEL
LIN {X 0,Y 291.632,Z 664.149,A -85,B 0,C 180,E1 -16569.712,E2 -16569.712} C_VEL
LIN {X 0,Y 291.524,Z 664.166,A -85,B 0,C 180,E1 -16573.95,E2 -16573.95} C_VEL
LIN {X 0,Y 291.489,Z 664.168,A -85,B 0,C 180,E1 -16576.818,E2 -16576.818} C_VEL
LIN {X 0,Y 291.453,Z 664.173,A -85,B 0,C 180,E1 -16579.875,E2 -16579.875} C_VEL
LIN {X 0,Y 291.402,Z 664.186,A -85,B 0,C 180,E1 -16584.205,E2 -16584.205} C_VEL
LIN {X 0,Y 291.421,Z 664.185,A -85,B 0,C 180,E1 -16587.272,E2 -16587.272} C_VEL
LIN {X 0,Y 291.337,Z 664.193,A -85,B 0,C 180,E1 -16590.437,E2 -16590.437} C_VEL
LIN {X 0,Y 291.347,Z 664.197,A -85,B 0,C 180,E1 -16593.698,E2 -16593.698} C_VEL
LIN {X 0,Y 291.418,Z 664.317,A -85,B 0,C 180,E1 -16596.647,E2 -16596.647} C_VEL
LIN {X 0,Y 292.586,Z 669.906,A -85,B 0,C 180,E1 -16600.433,E2 -16600.433} C_VEL
LIN {X 0,Y 293.777,Z 675.678,A -85,B 0,C 180,E1 -16603.929,E2 -16603.929} C_VEL
LIN {X 0,Y 295.057,Z 682.331,A -85,B 0,C 180,E1 -16607.595,E2 -16607.595} C_VEL
LIN {X 0,Y 296.175,Z 688.912,A -85,B 0,C 180,E1 -16610.925,E2 -16610.925} C_VEL
LIN {X 0,Y 296.18,Z 691.025,A -85,B 0,C 180,E1 -16611.906,E2 -16611.906} C_VEL
LIN {X 0,Y 294.544,Z 700.238,A -85,B 0,C 180,E1 -16615.894,E2 -16615.894} C_VEL
LIN {X 0,Y 292.876,Z 711.402,A -85,B 0,C 180,E1 -16620.532,E2 -16620.532} C_VEL
LIN {X 0,Y 292.084,Z 718.166,A -85,B 0,C 180,E1 -16623.259,E2 -16623.259} C_VEL
LIN {X 0,Y 295.024,Z 733.524,A -85,B 0,C 180,E1 -16624.319,E2 -16624.319} C_VEL
LIN {X 0,Y 296.636,Z 746.532,A -85,B 0,C 180,E1 -16625.394,E2 -16625.394} C_VEL
LIN {X 0,Y 297.254,Z 757.627,A -85,B 0,C 180,E1 -16626.46,E2 -16626.46} C_VEL
LIN {X 0,Y 297.088,Z 770.653,A -85,B 0,C 180,E1 -16627.942,E2 -16627.942} C_VEL
LIN {X 0,Y 297.205,Z 785.758,A -85,B 0,C 180,E1 -16629.224,E2 -16629.224} C_VEL
LIN {X 0,Y 296.856,Z 792.531,A -85,B 0,C 180,E1 -16629.922,E2 -16629.922} C_VEL
LIN {X 0,Y 295.385,Z 803.671,A -85,B 0,C 180,E1 -16631.264,E2 -16631.264} C_VEL
LIN {X 0,Y 294.199,Z 813.18,A -85,B 0,C 180,E1 -16632.697,E2 -16632.697} C_VEL
LIN {X 0,Y 293.028,Z 822.108,A -85,B 0,C 180,E1 -16634.346,E2 -16634.346} C_VEL
LIN {X 0,Y 291.696,Z 831.12,A -85,B 0,C 180,E1 -16636.413,E2 -16636.413} C_VEL
LIN {X 0,Y 290.753,Z 838.369,A -85,B 0,C 180,E1 -16638.496,E2 -16638.496} C_VEL
LIN {X 0,Y 290.207,Z 843.241,A -85,B 0,C 180,E1 -16640.239,E2 -16640.239} C_VEL
LIN {X 0,Y 289.818,Z 847.946,A -85,B 0,C 180,E1 -16642.335,E2 -16642.335} C_VEL
LIN {X 0,Y 289.586,Z 851.493,A -85,B 0,C 180,E1 -16644.428,E2 -16644.428} C_VEL
LIN {X 0,Y 289.537,Z 853.265,A -85,B 0,C 180,E1 -16645.823,E2 -16645.823} C_VEL
LIN {X 0,Y 289.537,Z 854.587,A -85,B 0,C 180,E1 -16647.217,E2 -16647.217} C_VEL
LIN {X 0,Y 289.513,Z 855.5,A -85,B 0,C 180,E1 -16648.608,E2 -16648.608} C_VEL
LIN {X 0,Y 289.547,Z 855.997,A -85,B 0,C 180,E1 -16649.999,E2 -16649.999} C_VEL
LIN {X 0,Y 289.502,Z 856.042,A -85,B 0,C 180,E1 -16651.39,E2 -16651.39} C_VEL
LIN {X 0,Y 289.53,Z 855.689,A -85,B 0,C 180,E1 -16652.782,E2 -16652.782} C_VEL
LIN {X 0,Y 289.505,Z 854.939,A -85,B 0,C 180,E1 -16654.176,E2 -16654.176} C_VEL
LIN {X 0,Y 289.552,Z 853.683,A -85,B 0,C 180,E1 -16655.641,E2 -16655.641} C_VEL
LIN {X 0,Y 289.935,Z 850.103,A -85,B 0,C 180,E1 -16658.362,E2 -16658.362} C_VEL
LIN {X 0,Y 290.537,Z 846.182,A -85,B 0,C 180,E1 -16660.452,E2 -16660.452} C_VEL
LIN {X 0,Y 291.387,Z 841.128,A -85,B 0,C 180,E1 -16662.536,E2 -16662.536} C_VEL
LIN {X 0,Y 292.726,Z 834.792,A -85,B 0,C 180,E1 -16664.6,E2 -16664.6} C_VEL
LIN {X 0,Y 294.317,Z 826.898,A -85,B 0,C 180,E1 -16666.65,E2 -16666.65} C_VEL
LIN {X 0,Y 295.814,Z 818.904,A -85,B 0,C 180,E1 -16668.348,E2 -16668.348} C_VEL
LIN {X 0,Y 297.649,Z 809.216,A -85,B 0,C 180,E1 -16670.02,E2 -16670.02} C_VEL
LIN {X 0,Y 299.671,Z 798.495,A -85,B 0,C 180,E1 -16671.496,E2 -16671.496} C_VEL
LIN {X 0,Y 300.764,Z 789.894,A -85,B 0,C 180,E1 -16672.496,E2 -16672.496} C_VEL
LIN {X 0,Y 301.226,Z 778.957,A -85,B 0,C 180,E1 -16673.6,E2 -16673.6} C_VEL
LIN {X 0,Y 301.339,Z 767.202,A -85,B 0,C 180,E1 -16674.552,E2 -16674.552} C_VEL
LIN {X 0,Y 300.242,Z 755.874,A -85,B 0,C 180,E1 -16675.363,E2 -16675.363} C_VEL
LIN {X 0,Y 297.302,Z 741.033,A -85,B 0,C 180,E1 -16676.33,E2 -16676.33} C_VEL
LIN {X 0,Y 296.509,Z 737.283,A -85,B 0,C 180,E1 -16676.621,E2 -16676.621} C_VEL
LIN {X 0,Y 295.422,Z 722.312,A -85,B 0,C 180,E1 -16678.992,E2 -16678.992} C_VEL
LIN {X 0,Y 294.492,Z 709.683,A -85,B 0,C 180,E1 -16681.293,E2 -16681.293} C_VEL
LIN {X 0,Y 293.985,Z 702.706,A -85,B 0,C 180,E1 -16682.728,E2 -16682.728} C_VEL
LIN {X 0,Y 295.761,Z 691.67,A -85,B 0,C 180,E1 -16687.295,E2 -16687.295} C_VEL
LIN {X 0,Y 296.031,Z 689.027,A -85,B 0,C 180,E1 -16688.423,E2 -16688.423} C_VEL
LIN {X 0,Y 295.442,Z 684.559,A -85,B 0,C 180,E1 -16690.428,E2 -16690.428} C_VEL
LIN {X 0,Y 293.84,Z 676.732,A -85,B 0,C 180,E1 -16694.148,E2 -16694.148} C_VEL
LIN {X 0,Y 292.3,Z 668.683,A -85,B 0,C 180,E1 -16698.188,E2 -16698.188} C_VEL
LIN {X 0,Y 291.417,Z 664.186,A -85,B 0,C 180,E1 -16700.63,E2 -16700.63} C_VEL
LIN {X 0,Y 291.426,Z 664.177,A -85,B 0,C 180,E1 -16702.922,E2 -16702.922} C_VEL
LIN {X 0,Y 291.341,Z 664.19,A -85,B 0,C 180,E1 -16706.301,E2 -16706.301} C_VEL
LIN {X 0,Y 291.383,Z 664.188,A -85,B 0,C 180,E1 -16710.259,E2 -16710.259} C_VEL
LIN {X 0,Y 291.412,Z 664.178,A -85,B 0,C 180,E1 -16714.271,E2 -16714.271} C_VEL
LIN {X 0,Y 291.385,Z 664.182,A -85,B 0,C 180,E1 -16717.3,E2 -16717.3} C_VEL
LIN {X 0,Y 291.455,Z 664.174,A -85,B 0,C 180,E1 -16720.27,E2 -16720.27} C_VEL
LIN {X 0,Y 291.512,Z 664.272,A -85,B 0,C 180,E1 -16723.382,E2 -16723.382} C_VEL
LIN {X 0,Y 292.798,Z 667.994,A -85,B 0,C 180,E1 -16726.112,E2 -16726.112} C_VEL
LIN {X 0,Y 294.554,Z 673.034,A -85,B 0,C 180,E1 -16729.407,E2 -16729.407} C_VEL
LIN {X 0,Y 296.297,Z 678.365,A -85,B 0,C 180,E1 -16732.504,E2 -16732.504} C_VEL
LIN {X 0,Y 298.158,Z 686.372,A -85,B 0,C 180,E1 -16736.621,E2 -16736.621} C_VEL
LIN {X 0,Y 299.173,Z 692.233,A -85,B 0,C 180,E1 -16739.327,E2 -16739.327} C_VEL
LIN {X 0,Y 299.486,Z 696.783,A -85,B 0,C 180,E1 -16741.344,E2 -16741.344} C_VEL
LIN {X 0,Y 298.932,Z 703.797,A -85,B 0,C 180,E1 -16744.044,E2 -16744.044} C_VEL
LIN {X 0,Y 297.496,Z 714.698,A -85,B 0,C 180,E1 -16748.149,E2 -16748.149} C_VEL
LIN {X 0,Y 296.417,Z 723.947,A -85,B 0,C 180,E1 -16751.626,E2 -16751.626} C_VEL
LIN {X 0,Y 295.595,Z 731.285,A -85,B 0,C 180,E1 -16754.368,E2 -16754.368} C_VEL
LIN {X 0,Y 299.483,Z 744.886,A -85,B 0,C 180,E1 -16755.508,E2 -16755.508} C_VEL
LIN {X 0,Y 301.775,Z 756.427,A -85,B 0,C 180,E1 -16756.576,E2 -16756.576} C_VEL
LIN {X 0,Y 302.959,Z 767.875,A -85,B 0,C 180,E1 -16757.757,E2 -16757.757} C_VEL
LIN {X 0,Y 301.949,Z 776.558,A -85,B 0,C 180,E1 -16758.63,E2 -16758.63} C_VEL
LIN {X 0,Y 300.098,Z 787.635,A -85,B 0,C 180,E1 -16759.977,E2 -16759.977} C_VEL
LIN {X 0,Y 298.055,Z 798.4,A -85,B 0,C 180,E1 -16761.619,E2 -16761.619} C_VEL
LIN {X 0,Y 296.113,Z 808.075,A -85,B 0,C 180,E1 -16763.491,E2 -16763.491} C_VEL
LIN {X 0,Y 294.397,Z 816.223,A -85,B 0,C 180,E1 -16765.449,E2 -16765.449} C_VEL
LIN {X 0,Y 292.947,Z 822.84,A -85,B 0,C 180,E1 -16767.423,E2 -16767.423} C_VEL
LIN {X 0,Y 291.601,Z 829.083,A -85,B 0,C 180,E1 -16769.816,E2 -16769.816} C_VEL
LIN {X 0,Y 290.627,Z 833.729,A -85,B 0,C 180,E1 -16772.182,E2 -16772.182} C_VEL
LIN {X 0,Y 289.907,Z 836.968,A -85,B 0,C 180,E1 -16774.491,E2 -16774.491} C_VEL
LIN {X 0,Y 289.426,Z 838.987,A -85,B 0,C 180,E1 -16776.745,E2 -16776.745} C_VEL
LIN {X 0,Y 289.172,Z 839.947,A -85,B 0,C 180,E1 -16779.19,E2 -16779.19} C_VEL
LIN {X 0,Y 289.056,Z 839.865,A -85,B 0,C 180,E1 -16781.088,E2 -16781.088} C_VEL
LIN {X 0,Y 289.103,Z 838.883,A -85,B 0,C 180,E1 -16783.175,E2 -16783.175} C_VEL
LIN {X 0,Y 289.284,Z 837.03,A -85,B 0,C 180,E1 -16785.209,E2 -16785.209} C_VEL
LIN {X 0,Y 289.64,Z 834.322,A -85,B 0,C 180,E1 -16787.204,E2 -16787.204} C_VEL
LIN {X 0,Y 290.043,Z 830.789,A -85,B 0,C 180,E1 -16789.14,E2 -16789.14} C_VEL
LIN {X 0,Y 290.848,Z 825.139,A -85,B 0,C 180,E1 -16791.506,E2 -16791.506} C_VEL
LIN {X 0,Y 291.852,Z 817.812,A -85,B 0,C 180,E1 -16793.846,E2 -16793.846} C_VEL
LIN {X 0,Y 293.067,Z 809.66,A -85,B 0,C 180,E1 -16795.907,E2 -16795.907} C_VEL
LIN {X 0,Y 294.348,Z 800.795,A -85,B 0,C 180,E1 -16797.709,E2 -16797.709} C_VEL
LIN {X 0,Y 295.873,Z 789.885,A -85,B 0,C 180,E1 -16799.488,E2 -16799.488} C_VEL
LIN {X 0,Y 297.343,Z 778.222,A -85,B 0,C 180,E1 -16800.99,E2 -16800.99} C_VEL
LIN {X 0,Y 298.738,Z 765.879,A -85,B 0,C 180,E1 -16802.22,E2 -16802.22} C_VEL
LIN {X 0,Y 297.624,Z 755.429,A -85,B 0,C 180,E1 -16803.154,E2 -16803.154} C_VEL
LIN {X 0,Y 295.549,Z 742.386,A -85,B 0,C 180,E1 -16804.092,E2 -16804.092} C_VEL
LIN {X 0,Y 293.304,Z 730.23,A -85,B 0,C 180,E1 -16804.752,E2 -16804.752} C_VEL
LIN {X 0,Y 294.264,Z 718.531,A -85,B 0,C 180,E1 -16809.008,E2 -16809.008} C_VEL
LIN {X 0,Y 295.125,Z 707.966,A -85,B 0,C 180,E1 -16812.87,E2 -16812.87} C_VEL
LIN {X 0,Y 296.093,Z 696.479,A -85,B 0,C 180,E1 -16817.07,E2 -16817.07} C_VEL
LIN {X 0,Y 296.417,Z 691.085,A -85,B 0,C 180,E1 -16819.067,E2 -16819.067} C_VEL
LIN {X 0,Y 295.967,Z 685.793,A -85,B 0,C 180,E1 -16821.122,E2 -16821.122} C_VEL
LIN {X 0,Y 294.838,Z 679.01,A -85,B 0,C 180,E1 -16823.843,E2 -16823.843} C_VEL
LIN {X 0,Y 292.584,Z 667.434,A -85,B 0,C 180,E1 -16828.624,E2 -16828.624} C_VEL
LIN {X 0,Y 291.964,Z 664.118,A -85,B 0,C 180,E1 -16830.087,E2 -16830.087} C_VEL
LIN {X 0,Y 291.8,Z 664.139,A -85,B 0,C 180,E1 -16832.762,E2 -16832.762} C_VEL
LIN {X 0,Y 291.743,Z 664.14,A -85,B 0,C 180,E1 -16836.919,E2 -16836.919} C_VEL
LIN {X 0,Y 291.631,Z 664.152,A -85,B 0,C 180,E1 -16839.712,E2 -16839.712} C_VEL
LIN {X 0,Y 291.52,Z 664.173,A -85,B 0,C 180,E1 -16843.951,E2 -16843.951} C_VEL
LIN {X 0,Y 291.57,Z 664.222,A -85,B 0,C 180,E1 -16845.207,E2 -16845.207} C_VEL
LIN {X 0,Y 295.267,Z 675.545,A -85,B 0,C 180,E1 -16846.419,E2 -16846.419} C_VEL
LIN {X 0,Y 298.474,Z 686.592,A -85,B 0,C 180,E1 -16847.825,E2 -16847.825} C_VEL
LIN {X 0,Y 299.558,Z 690.8,A -85,B 0,C 180,E1 -16848.427,E2 -16848.427} C_VEL
LIN {X 0,Y 298.496,Z 701.821,A -85,B 0,C 180,E1 -16849.933,E2 -16849.933} C_VEL
LIN {X 0,Y 297.17,Z 712.12,A -85,B 0,C 180,E1 -16851.687,E2 -16851.687} C_VEL
LIN {X 0,Y 296.003,Z 720.556,A -85,B 0,C 180,E1 -16853.454,E2 -16853.454} C_VEL
LIN {X 0,Y 294.889,Z 728.153,A -85,B 0,C 180,E1 -16855.404,E2 -16855.404} C_VEL
LIN {X 0,Y 293.784,Z 735.323,A -85,B 0,C 180,E1 -16857.733,E2 -16857.733} C_VEL
LIN {X 0,Y 292.954,Z 741.31,A -85,B 0,C 180,E1 -16860.272,E2 -16860.272} C_VEL
LIN {X 0,Y 292.263,Z 745.438,A -85,B 0,C 180,E1 -16862.686,E2 -16862.686} C_VEL
LIN {X 0,Y 291.857,Z 748.424,A -85,B 0,C 180,E1 -16865.305,E2 -16865.305} C_VEL
LIN {X 0,Y 291.78,Z 749.731,A -85,B 0,C 180,E1 -16867.358,E2 -16867.358} C_VEL
LIN {X 0,Y 291.949,Z 750.167,A -85,B 0,C 180,E1 -16869.617,E2 -16869.617} C_VEL
LIN {X 0,Y 292.448,Z 749.347,A -85,B 0,C 180,E1 -16872.291,E2 -16872.291} C_VEL
LIN {X 0,Y 293.24,Z 746.956,A -85,B 0,C 180,E1 -16874.993,E2 -16874.993} C_VEL
LIN {X 0,Y 294.456,Z 742.874,A -85,B 0,C 180,E1 -16877.724,E2 -16877.724} C_VEL
LIN {X 0,Y 295.736,Z 737.794,A -85,B 0,C 180,E1 -16880.086,E2 -16880.086} C_VEL
LIN {X 0,Y 297.082,Z 732.321,A -85,B 0,C 180,E1 -16882.043,E2 -16882.043} C_VEL
LIN {X 0,Y 298.737,Z 724.945,A -85,B 0,C 180,E1 -16884.14,E2 -16884.14} C_VEL
LIN {X 0,Y 300.517,Z 715.863,A -85,B 0,C 180,E1 -16886.169,E2 -16886.169} C_VEL
LIN {X 0,Y 302.335,Z 706.226,A -85,B 0,C 180,E1 -16887.877,E2 -16887.877} C_VEL
LIN {X 0,Y 303.557,Z 697.322,A -85,B 0,C 180,E1 -16889.181,E2 -16889.181} C_VEL
LIN {X 0,Y 300.916,Z 687.711,A -85,B 0,C 180,E1 -16890.771,E2 -16890.771} C_VEL
LIN {X 0,Y 297.383,Z 677.831,A -85,B 0,C 180,E1 -16892.257,E2 -16892.257} C_VEL
LIN {X 0,Y 292.883,Z 667.658,A -85,B 0,C 180,E1 -16893.69,E2 -16893.69} C_VEL
LIN {X 0,Y 290.936,Z 665.852,A -85,B 0,C 180,E1 -16894.21,E2 -16894.21} C_VEL
LIN {X 0,Y 288.76,Z 664.873,A -85,B 0,C 180,E1 -16895.028,E2 -16895.028} C_VEL
LIN {X 0,Y 286.446,Z 664.796,A -85,B 0,C 180,E1 -16896.32,E2 -16896.32} C_VEL
LIN {X 0,Y 284.816,Z 664.999,A -85,B 0,C 180,E1 -16897.973,E2 -16897.973} C_VEL
LIN {X 0,Y 284.37,Z 665.064,A -85,B 0,C 180,E1 -16899.662,E2 -16899.662} C_VEL
LIN {X 0,Y 284.49,Z 665.052,A -85,B 0,C 180,E1 -16904.232,E2 -16904.232} C_VEL
LIN {X 0,Y 284.49,Z 665.041,A -85,B 0,C 180,E1 -16908.602,E2 -16908.602} C_VEL
LIN {X 0,Y 284.661,Z 665.021,A -85,B 0,C 180,E1 -16911.481,E2 -16911.481} C_VEL
LIN {X 0,Y 284.604,Z 665.035,A -85,B 0,C 180,E1 -16914.332,E2 -16914.332} C_VEL
LIN {X 0,Y 284.858,Z 665.001,A -85,B 0,C 180,E1 -16918.586,E2 -16918.586} C_VEL
LIN {X 0,Y 284.858,Z 664.99,A -85,B 0,C 180,E1 -16921.414,E2 -16921.414} C_VEL
LIN {X 0,Y 284.701,Z 665.021,A -85,B 0,C 180,E1 -16927.09,E2 -16927.09} C_VEL
LIN {X 0,Y 284.569,Z 665.031,A -85,B 0,C 180,E1 -16929.955,E2 -16929.955} C_VEL
LIN {X 0,Y 284.484,Z 665.046,A -85,B 0,C 180,E1 -16934.303,E2 -16934.303} C_VEL
LIN {X 0,Y 284.428,Z 665.049,A -85,B 0,C 180,E1 -16937.248,E2 -16937.248} C_VEL
LIN {X 0,Y 284.381,Z 665.055,A -85,B 0,C 180,E1 -16940.242,E2 -16940.242} C_VEL
LIN {X 0,Y 284.371,Z 665.06,A -85,B 0,C 180,E1 -16943.875,E2 -16943.875} C_VEL
LIN {X 0,Y 284.397,Z 665.06,A -85,B 0,C 180,E1 -16947.172,E2 -16947.172} C_VEL
LIN {X 0,Y 284.296,Z 665.072,A -85,B 0,C 180,E1 -16951.275,E2 -16951.275} C_VEL
LIN {X 0,Y 284.349,Z 665.156,A -85,B 0,C 180,E1 -16955.652,E2 -16955.652} C_VEL
LIN {X 0,Y 285.575,Z 670.958,A -85,B 0,C 180,E1 -16959.782,E2 -16959.782} C_VEL
LIN {X 0,Y 286.772,Z 676.578,A -85,B 0,C 180,E1 -16963.331,E2 -16963.331} C_VEL
LIN {X 0,Y 288.009,Z 683.095,A -85,B 0,C 180,E1 -16967.06,E2 -16967.06} C_VEL
LIN {X 0,Y 288.99,Z 688.492,A -85,B 0,C 180,E1 -16969.922,E2 -16969.922} C_VEL
LIN {X 0,Y 289.195,Z 692.354,A -85,B 0,C 180,E1 -16971.808,E2 -16971.808} C_VEL
LIN {X 0,Y 287.342,Z 702.423,A -85,B 0,C 180,E1 -16976.263,E2 -16976.263} C_VEL
LIN {X 0,Y 285.609,Z 714.315,A -85,B 0,C 180,E1 -16981.325,E2 -16981.325} C_VEL
LIN {X 0,Y 285.27,Z 716.954,A -85,B 0,C 180,E1 -16982.414,E2 -16982.414} C_VEL
LIN {X 0,Y 288.206,Z 731.705,A -85,B 0,C 180,E1 -16983.476,E2 -16983.476} C_VEL
LIN {X 0,Y 289.937,Z 744.71,A -85,B 0,C 180,E1 -16984.592,E2 -16984.592} C_VEL
LIN {X 0,Y 290.637,Z 757.71,A -85,B 0,C 180,E1 -16985.904,E2 -16985.904} C_VEL
LIN {X 0,Y 290.405,Z 770.37,A -85,B 0,C 180,E1 -16987.406,E2 -16987.406} C_VEL
LIN {X 0,Y 290.27,Z 773.558,A -85,B 0,C 180,E1 -16987.77,E2 -16987.77} C_VEL
LIN {X 0,Y 290.32,Z 786.23,A -85,B 0,C 180,E1 -16988.894,E2 -16988.894} C_VEL
LIN {X 0,Y 289.949,Z 792.91,A -85,B 0,C 180,E1 -16989.608,E2 -16989.608} C_VEL
LIN {X 0,Y 288.451,Z 803.942,A -85,B 0,C 180,E1 -16990.981,E2 -16990.981} C_VEL
LIN {X 0,Y 287.089,Z 814.332,A -85,B 0,C 180,E1 -16992.619,E2 -16992.619} C_VEL
LIN {X 0,Y 285.889,Z 823.022,A -85,B 0,C 180,E1 -16994.311,E2 -16994.311} C_VEL
LIN {X 0,Y 284.552,Z 831.849,A -85,B 0,C 180,E1 -16996.429,E2 -16996.429} C_VEL
LIN {X 0,Y 283.621,Z 838.885,A -85,B 0,C 180,E1 -16998.565,E2 -16998.565} C_VEL
LIN {X 0,Y 282.998,Z 844.478,A -85,B 0,C 180,E1 -17000.71,E2 -17000.71} C_VEL
LIN {X 0,Y 282.66,Z 848.839,A -85,B 0,C 180,E1 -17002.858,E2 -17002.858} C_VEL
LIN {X 0,Y 282.524,Z 851.128,A -85,B 0,C 180,E1 -17004.289,E2 -17004.289} C_VEL
LIN {X 0,Y 282.44,Z 852.952,A -85,B 0,C 180,E1 -17005.718,E2 -17005.718} C_VEL
LIN {X 0,Y 282.463,Z 854.3,A -85,B 0,C 180,E1 -17007.147,E2 -17007.147} C_VEL
LIN {X 0,Y 282.433,Z 855.237,A -85,B 0,C 180,E1 -17008.573,E2 -17008.573} C_VEL
LIN {X 0,Y 282.462,Z 855.771,A -85,B 0,C 180,E1 -17009.999,E2 -17009.999} C_VEL
LIN {X 0,Y 282.421,Z 855.851,A -85,B 0,C 180,E1 -17011.425,E2 -17011.425} C_VEL
LIN {X 0,Y 282.433,Z 855.521,A -85,B 0,C 180,E1 -17012.852,E2 -17012.852} C_VEL
LIN {X 0,Y 282.462,Z 853.784,A -85,B 0,C 180,E1 -17015.584,E2 -17015.584} C_VEL
LIN {X 0,Y 282.751,Z 851.158,A -85,B 0,C 180,E1 -17017.857,E2 -17017.857} C_VEL
LIN {X 0,Y 283.316,Z 847.648,A -85,B 0,C 180,E1 -17019.999,E2 -17019.999} C_VEL
LIN {X 0,Y 284.146,Z 843.046,A -85,B 0,C 180,E1 -17022.135,E2 -17022.135} C_VEL
LIN {X 0,Y 285.602,Z 836.089,A -85,B 0,C 180,E1 -17024.609,E2 -17024.609} C_VEL
LIN {X 0,Y 287.26,Z 828.608,A -85,B 0,C 180,E1 -17026.706,E2 -17026.706} C_VEL
LIN {X 0,Y 288.745,Z 821.053,A -85,B 0,C 180,E1 -17028.445,E2 -17028.445} C_VEL
LIN {X 0,Y 290.819,Z 810.871,A -85,B 0,C 180,E1 -17030.327,E2 -17030.327} C_VEL
LIN {X 0,Y 293.132,Z 799.353,A -85,B 0,C 180,E1 -17032,E2 -17032} C_VEL
LIN {X 0,Y 294.284,Z 790.896,A -85,B 0,C 180,E1 -17033.02,E2 -17033.02} C_VEL
LIN {X 0,Y 294.872,Z 779.925,A -85,B 0,C 180,E1 -17034.182,E2 -17034.182} C_VEL
LIN {X 0,Y 295.053,Z 767.073,A -85,B 0,C 180,E1 -17035.269,E2 -17035.269} C_VEL
LIN {X 0,Y 293.826,Z 755.296,A -85,B 0,C 180,E1 -17036.165,E2 -17036.165} C_VEL
LIN {X 0,Y 291.177,Z 742.023,A -85,B 0,C 180,E1 -17037.077,E2 -17037.077} C_VEL
LIN {X 0,Y 290.114,Z 737.623,A -85,B 0,C 180,E1 -17037.404,E2 -17037.404} C_VEL
LIN {X 0,Y 289.291,Z 724.009,A -85,B 0,C 180,E1 -17039.667,E2 -17039.667} C_VEL
LIN {X 0,Y 288.438,Z 711.64,A -85,B 0,C 180,E1 -17042.036,E2 -17042.036} C_VEL
LIN {X 0,Y 288,Z 704.719,A -85,B 0,C 180,E1 -17043.496,E2 -17043.496} C_VEL
LIN {X 0,Y 287.795,Z 697.896,A -85,B 0,C 180,E1 -17045.126,E2 -17045.126} C_VEL
LIN {X 0,Y 289.014,Z 690.784,A -85,B 0,C 180,E1 -17048.169,E2 -17048.169} C_VEL
LIN {X 0,Y 288.945,Z 688.423,A -85,B 0,C 180,E1 -17049.226,E2 -17049.226} C_VEL
LIN {X 0,Y 287.45,Z 680.893,A -85,B 0,C 180,E1 -17052.82,E2 -17052.82} C_VEL
LIN {X 0,Y 285.778,Z 672.322,A -85,B 0,C 180,E1 -17057.143,E2 -17057.143} C_VEL
LIN {X 0,Y 284.354,Z 665.066,A -85,B 0,C 180,E1 -17061.074,E2 -17061.074} C_VEL
LIN {X 0,Y 284.359,Z 665.058,A -85,B 0,C 180,E1 -17064.645,E2 -17064.645} C_VEL
LIN {X 0,Y 284.292,Z 665.064,A -85,B 0,C 180,E1 -17068.725,E2 -17068.725} C_VEL
LIN {X 0,Y 284.393,Z 665.062,A -85,B 0,C 180,E1 -17072.826,E2 -17072.826} C_VEL
LIN {X 0,Y 284.364,Z 665.057,A -85,B 0,C 180,E1 -17076.707,E2 -17076.707} C_VEL
LIN {X 0,Y 284.431,Z 665.095,A -85,B 0,C 180,E1 -17080.242,E2 -17080.242} C_VEL
LIN {X 0,Y 286.069,Z 669.701,A -85,B 0,C 180,E1 -17084.321,E2 -17084.321} C_VEL
LIN {X 0,Y 287.706,Z 674.279,A -85,B 0,C 180,E1 -17087.712,E2 -17087.712} C_VEL
LIN {X 0,Y 289.39,Z 679.272,A -85,B 0,C 180,E1 -17090.917,E2 -17090.917} C_VEL
LIN {X 0,Y 290.415,Z 682.95,A -85,B 0,C 180,E1 -17093.05,E2 -17093.05} C_VEL
LIN {X 0,Y 292.115,Z 691.05,A -85,B 0,C 180,E1 -17097.242,E2 -17097.242} C_VEL
LIN {X 0,Y 292.736,Z 695.352,A -85,B 0,C 180,E1 -17099.312,E2 -17099.312} C_VEL
LIN {X 0,Y 292.998,Z 700.089,A -85,B 0,C 180,E1 -17101.374,E2 -17101.374} C_VEL
LIN {X 0,Y 292.243,Z 707.074,A -85,B 0,C 180,E1 -17104.137,E2 -17104.137} C_VEL
LIN {X 0,Y 290.713,Z 717.971,A -85,B 0,C 180,E1 -17108.34,E2 -17108.34} C_VEL
LIN {X 0,Y 289.574,Z 727.277,A -85,B 0,C 180,E1 -17111.905,E2 -17111.905} C_VEL
LIN {X 0,Y 289.048,Z 731.628,A -85,B 0,C 180,E1 -17113.525,E2 -17113.525} C_VEL
LIN {X 0,Y 292.696,Z 743.892,A -85,B 0,C 180,E1 -17114.603,E2 -17114.603} C_VEL
LIN {X 0,Y 295.109,Z 755.372,A -85,B 0,C 180,E1 -17115.708,E2 -17115.708} C_VEL
LIN {X 0,Y 296.47,Z 766.375,A -85,B 0,C 180,E1 -17116.881,E2 -17116.881} C_VEL
LIN {X 0,Y 296.547,Z 771.193,A -85,B 0,C 180,E1 -17117.41,E2 -17117.41} C_VEL
LIN {X 0,Y 294.6,Z 782.997,A -85,B 0,C 180,E1 -17118.715,E2 -17118.715} C_VEL
LIN {X 0,Y 292.692,Z 793.256,A -85,B 0,C 180,E1 -17120.149,E2 -17120.149} C_VEL
LIN {X 0,Y 290.704,Z 802.904,A -85,B 0,C 180,E1 -17121.821,E2 -17121.821} C_VEL
LIN {X 0,Y 288.813,Z 811.471,A -85,B 0,C 180,E1 -17123.673,E2 -17123.673} C_VEL
LIN {X 0,Y 287.148,Z 818.838,A -85,B 0,C 180,E1 -17125.64,E2 -17125.64} C_VEL
LIN {X 0,Y 285.532,Z 825.595,A -85,B 0,C 180,E1 -17127.882,E2 -17127.882} C_VEL
LIN {X 0,Y 284.373,Z 830.809,A -85,B 0,C 180,E1 -17130.121,E2 -17130.121} C_VEL
LIN {X 0,Y 283.414,Z 835.003,A -85,B 0,C 180,E1 -17132.531,E2 -17132.531} C_VEL
LIN {X 0,Y 282.715,Z 837.86,A -85,B 0,C 180,E1 -17134.882,E2 -17134.882} C_VEL
LIN {X 0,Y 282.303,Z 839.555,A -85,B 0,C 180,E1 -17137.191,E2 -17137.191} C_VEL
LIN {X 0,Y 282.071,Z 840.187,A -85,B 0,C 180,E1 -17139.433,E2 -17139.433} C_VEL
LIN {X 0,Y 281.949,Z 839.565,A -85,B 0,C 180,E1 -17142.3,E2 -17142.3} C_VEL
LIN {X 0,Y 282.081,Z 838.21,A -85,B 0,C 180,E1 -17144.236,E2 -17144.236} C_VEL
LIN {X 0,Y 282.518,Z 834.865,A -85,B 0,C 180,E1 -17147.02,E2 -17147.02} C_VEL
LIN {X 0,Y 282.933,Z 831.433,A -85,B 0,C 180,E1 -17149.009,E2 -17149.009} C_VEL
LIN {X 0,Y 283.548,Z 826.958,A -85,B 0,C 180,E1 -17151.021,E2 -17151.021} C_VEL
LIN {X 0,Y 284.503,Z 820.387,A -85,B 0,C 180,E1 -17153.336,E2 -17153.336} C_VEL
LIN {X 0,Y 285.655,Z 812.468,A -85,B 0,C 180,E1 -17155.538,E2 -17155.538} C_VEL
LIN {X 0,Y 286.931,Z 804.117,A -85,B 0,C 180,E1 -17157.395,E2 -17157.395} C_VEL
LIN {X 0,Y 288.463,Z 793.949,A -85,B 0,C 180,E1 -17159.228,E2 -17159.228} C_VEL
LIN {X 0,Y 289.913,Z 783.207,A -85,B 0,C 180,E1 -17160.774,E2 -17160.774} C_VEL
LIN {X 0,Y 291.4,Z 771.13,A -85,B 0,C 180,E1 -17162.143,E2 -17162.143} C_VEL
LIN {X 0,Y 291.911,Z 766.43,A -85,B 0,C 180,E1 -17162.585,E2 -17162.585} C_VEL
LIN {X 0,Y 290.572,Z 754.758,A -85,B 0,C 180,E1 -17163.662,E2 -17163.662} C_VEL
LIN {X 0,Y 288.357,Z 740.915,A -85,B 0,C 180,E1 -17164.658,E2 -17164.658} C_VEL
LIN {X 0,Y 286.397,Z 730.408,A -85,B 0,C 180,E1 -17165.224,E2 -17165.224} C_VEL
LIN {X 0,Y 287.347,Z 719.533,A -85,B 0,C 180,E1 -17169.229,E2 -17169.229} C_VEL
LIN {X 0,Y 288.296,Z 708.398,A -85,B 0,C 180,E1 -17173.356,E2 -17173.356} C_VEL
LIN {X 0,Y 289.227,Z 697.614,A -85,B 0,C 180,E1 -17177.369,E2 -17177.369} C_VEL
LIN {X 0,Y 289.534,Z 691.936,A -85,B 0,C 180,E1 -17179.512,E2 -17179.512} C_VEL
LIN {X 0,Y 288.738,Z 684.929,A -85,B 0,C 180,E1 -17182.307,E2 -17182.307} C_VEL
LIN {X 0,Y 287.447,Z 678.209,A -85,B 0,C 180,E1 -17185.092,E2 -17185.092} C_VEL
LIN {X 0,Y 285.602,Z 668.21,A -85,B 0,C 180,E1 -17189.296,E2 -17189.296} C_VEL
LIN {X 0,Y 284.887,Z 665,A -85,B 0,C 180,E1 -17190.707,E2 -17190.707} C_VEL
LIN {X 0,Y 284.752,Z 665.017,A -85,B 0,C 180,E1 -17192.83,E2 -17192.83} C_VEL
LIN {X 0,Y 284.695,Z 665.018,A -85,B 0,C 180,E1 -17197.091,E2 -17197.091} C_VEL
LIN {X 0,Y 284.568,Z 665.032,A -85,B 0,C 180,E1 -17199.956,E2 -17199.956} C_VEL
LIN {X 0,Y 284.513,Z 665.189,A -85,B 0,C 180,E1 -17204.713,E2 -17204.713} C_VEL
LIN {X 0,Y 288.575,Z 677.457,A -85,B 0,C 180,E1 -17206.084,E2 -17206.084} C_VEL
LIN {X 0,Y 291.566,Z 687.809,A -85,B 0,C 180,E1 -17207.447,E2 -17207.447} C_VEL
LIN {X 0,Y 292.777,Z 692.864,A -85,B 0,C 180,E1 -17208.184,E2 -17208.184} C_VEL
LIN {X 0,Y 291.603,Z 703.633,A -85,B 0,C 180,E1 -17209.72,E2 -17209.72} C_VEL
LIN {X 0,Y 290.269,Z 713.631,A -85,B 0,C 180,E1 -17211.482,E2 -17211.482} C_VEL
LIN {X 0,Y 289.069,Z 721.906,A -85,B 0,C 180,E1 -17213.272,E2 -17213.272} C_VEL
LIN {X 0,Y 287.842,Z 729.838,A -85,B 0,C 180,E1 -17215.392,E2 -17215.392} C_VEL
LIN {X 0,Y 286.731,Z 736.824,A -85,B 0,C 180,E1 -17217.756,E2 -17217.756} C_VEL
LIN {X 0,Y 285.969,Z 742.018,A -85,B 0,C 180,E1 -17220.018,E2 -17220.018} C_VEL
LIN {X 0,Y 285.434,Z 745.45,A -85,B 0,C 180,E1 -17221.964,E2 -17221.964} C_VEL
LIN {X 0,Y 284.917,Z 748.771,A -85,B 0,C 180,E1 -17224.565,E2 -17224.565} C_VEL
LIN {X 0,Y 284.768,Z 750.18,A -85,B 0,C 180,E1 -17226.322,E2 -17226.322} C_VEL
LIN {X 0,Y 284.78,Z 751.012,A -85,B 0,C 180,E1 -17228.096,E2 -17228.096} C_VEL
LIN {X 0,Y 285.019,Z 751.203,A -85,B 0,C 180,E1 -17230.147,E2 -17230.147} C_VEL
LIN {X 0,Y 285.478,Z 750.453,A -85,B 0,C 180,E1 -17232.392,E2 -17232.392} C_VEL
LIN {X 0,Y 286.094,Z 748.77,A -85,B 0,C 180,E1 -17234.57,E2 -17234.57} C_VEL
LIN {X 0,Y 287.209,Z 745.304,A -85,B 0,C 180,E1 -17237.232,E2 -17237.232} C_VEL
LIN {X 0,Y 288.17,Z 741.885,A -85,B 0,C 180,E1 -17239.117,E2 -17239.117} C_VEL
LIN {X 0,Y 289.681,Z 736.314,A -85,B 0,C 180,E1 -17241.452,E2 -17241.452} C_VEL
LIN {X 0,Y 291.09,Z 730.424,A -85,B 0,C 180,E1 -17243.397,E2 -17243.397} C_VEL
LIN {X 0,Y 292.778,Z 723.281,A -85,B 0,C 180,E1 -17245.289,E2 -17245.289} C_VEL
LIN {X 0,Y 294.415,Z 715.249,A -85,B 0,C 180,E1 -17247.028,E2 -17247.028} C_VEL
LIN {X 0,Y 296.191,Z 705.786,A -85,B 0,C 180,E1 -17248.673,E2 -17248.673} C_VEL
LIN {X 0,Y 297.132,Z 699.712,A -85,B 0,C 180,E1 -17249.567,E2 -17249.567} C_VEL
LIN {X 0,Y 294.556,Z 690.108,A -85,B 0,C 180,E1 -17251.24,E2 -17251.24} C_VEL
LIN {X 0,Y 291.354,Z 680.866,A -85,B 0,C 180,E1 -17252.722,E2 -17252.722} C_VEL
LIN {X 0,Y 286.921,Z 670.94,A -85,B 0,C 180,E1 -17254.229,E2 -17254.229} C_VEL
LIN {X 0,Y 284.552,Z 666.042,A -85,B 0,C 180,E1 -17254.93,E2 -17254.93} C_VEL
LIN {X 0,Y 284.335,Z 665.067,A -85,B 0,C 180,E1 -17255.056,E2 -17255.056} C_VEL
LIN {X 0,Y 284.37,Z 665.064,A -85,B 0,C 180,E1 -17259.662,E2 -17259.662} C_VEL
LIN {X 0,Y 283.793,Z 665.146,A -85,B 0,C 180,E1 -17260.845,E2 -17260.845} C_VEL
LIN {X 0,Y 280.992,Z 665.494,A -85,B 0,C 180,E1 -17262.773,E2 -17262.773} C_VEL
LIN {X 0,Y 278.555,Z 665.791,A -85,B 0,C 180,E1 -17264.338,E2 -17264.338} C_VEL
LIN {X 0,Y 277.496,Z 665.917,A -85,B 0,C 180,E1 -17265.552,E2 -17265.552} C_VEL
LIN {X 0,Y 277.406,Z 665.927,A -85,B 0,C 180,E1 -17265.963,E2 -17265.963} C_VEL
LIN {X 0,Y 277.633,Z 665.901,A -85,B 0,C 180,E1 -17270.841,E2 -17270.841} C_VEL
LIN {X 0,Y 277.574,Z 665.909,A -85,B 0,C 180,E1 -17274.187,E2 -17274.187} C_VEL
LIN {X 0,Y 277.824,Z 665.878,A -85,B 0,C 180,E1 -17278.551,E2 -17278.551} C_VEL
LIN {X 0,Y 277.824,Z 665.866,A -85,B 0,C 180,E1 -17281.45,E2 -17281.45} C_VEL
LIN {X 0,Y 277.656,Z 665.898,A -85,B 0,C 180,E1 -17287.271,E2 -17287.271} C_VEL
LIN {X 0,Y 277.509,Z 665.912,A -85,B 0,C 180,E1 -17290.211,E2 -17290.211} C_VEL
LIN {X 0,Y 277.437,Z 665.927,A -85,B 0,C 180,E1 -17294.674,E2 -17294.674} C_VEL
LIN {X 0,Y 277.348,Z 665.933,A -85,B 0,C 180,E1 -17299.234,E2 -17299.234} C_VEL
LIN {X 0,Y 277.321,Z 665.94,A -85,B 0,C 180,E1 -17304.17,E2 -17304.17} C_VEL
LIN {X 0,Y 277.325,Z 665.94,A -85,B 0,C 180,E1 -17307.504,E2 -17307.504} C_VEL
LIN {X 0,Y 277.275,Z 665.944,A -85,B 0,C 180,E1 -17310.481,E2 -17310.481} C_VEL
LIN {X 0,Y 277.258,Z 665.949,A -85,B 0,C 180,E1 -17314.553,E2 -17314.553} C_VEL
LIN {X 0,Y 278.406,Z 671.188,A -85,B 0,C 180,E1 -17318.504,E2 -17318.504} C_VEL
LIN {X 0,Y 279.736,Z 677.498,A -85,B 0,C 180,E1 -17322.714,E2 -17322.714} C_VEL
LIN {X 0,Y 280.954,Z 683.843,A -85,B 0,C 180,E1 -17326.505,E2 -17326.505} C_VEL
LIN {X 0,Y 281.974,Z 689.511,A -85,B 0,C 180,E1 -17329.606,E2 -17329.606} C_VEL
LIN {X 0,Y 282.275,Z 693.287,A -85,B 0,C 180,E1 -17331.505,E2 -17331.505} C_VEL
LIN {X 0,Y 280.48,Z 702.614,A -85,B 0,C 180,E1 -17335.78,E2 -17335.78} C_VEL
LIN {X 0,Y 278.755,Z 713.48,A -85,B 0,C 180,E1 -17340.551,E2 -17340.551} C_VEL
LIN {X 0,Y 278.513,Z 715.816,A -85,B 0,C 180,E1 -17341.497,E2 -17341.497} C_VEL
LIN {X 0,Y 281.563,Z 730.735,A -85,B 0,C 180,E1 -17342.654,E2 -17342.654} C_VEL
LIN {X 0,Y 283.286,Z 743.638,A -85,B 0,C 180,E1 -17343.81,E2 -17343.81} C_VEL
LIN {X 0,Y 284.029,Z 756.212,A -85,B 0,C 180,E1 -17345.124,E2 -17345.124} C_VEL
LIN {X 0,Y 283.817,Z 768.751,A -85,B 0,C 180,E1 -17346.659,E2 -17346.659} C_VEL
LIN {X 0,Y 283.475,Z 774.289,A -85,B 0,C 180,E1 -17347.4,E2 -17347.4} C_VEL
LIN {X 0,Y 283.465,Z 786.678,A -85,B 0,C 180,E1 -17348.549,E2 -17348.549} C_VEL
LIN {X 0,Y 283.053,Z 793.283,A -85,B 0,C 180,E1 -17349.278,E2 -17349.278} C_VEL
LIN {X 0,Y 281.522,Z 804.212,A -85,B 0,C 180,E1 -17350.683,E2 -17350.683} C_VEL
LIN {X 0,Y 280.301,Z 813.132,A -85,B 0,C 180,E1 -17352.112,E2 -17352.112} C_VEL
LIN {X 0,Y 279.033,Z 822.311,A -85,B 0,C 180,E1 -17353.915,E2 -17353.915} C_VEL
LIN {X 0,Y 277.618,Z 831.222,A -85,B 0,C 180,E1 -17356.083,E2 -17356.083} C_VEL
LIN {X 0,Y 276.603,Z 838.363,A -85,B 0,C 180,E1 -17358.271,E2 -17358.271} C_VEL
LIN {X 0,Y 275.96,Z 844.021,A -85,B 0,C 180,E1 -17360.471,E2 -17360.471} C_VEL
LIN {X 0,Y 275.598,Z 848.44,A -85,B 0,C 180,E1 -17362.674,E2 -17362.674} C_VEL
LIN {X 0,Y 275.436,Z 851.043,A -85,B 0,C 180,E1 -17364.34,E2 -17364.34} C_VEL
LIN {X 0,Y 275.348,Z 852.623,A -85,B 0,C 180,E1 -17365.608,E2 -17365.608} C_VEL
LIN {X 0,Y 275.367,Z 854.006,A -85,B 0,C 180,E1 -17367.073,E2 -17367.073} C_VEL
LIN {X 0,Y 275.354,Z 854.968,A -85,B 0,C 180,E1 -17368.537,E2 -17368.537} C_VEL
LIN {X 0,Y 275.379,Z 855.53,A -85,B 0,C 180,E1 -17369.999,E2 -17369.999} C_VEL
LIN {X 0,Y 275.343,Z 855.662,A -85,B 0,C 180,E1 -17371.462,E2 -17371.462} C_VEL
LIN {X 0,Y 275.339,Z 855.36,A -85,B 0,C 180,E1 -17372.925,E2 -17372.925} C_VEL
LIN {X 0,Y 275.394,Z 853.572,A -85,B 0,C 180,E1 -17375.858,E2 -17375.858} C_VEL
LIN {X 0,Y 275.58,Z 852.032,A -85,B 0,C 180,E1 -17377.325,E2 -17377.325} C_VEL
LIN {X 0,Y 276.08,Z 848.922,A -85,B 0,C 180,E1 -17379.523,E2 -17379.523} C_VEL
LIN {X 0,Y 276.86,Z 844.755,A -85,B 0,C 180,E1 -17381.716,E2 -17381.716} C_VEL
LIN {X 0,Y 278.181,Z 838.431,A -85,B 0,C 180,E1 -17384.259,E2 -17384.259} C_VEL
LIN {X 0,Y 279.88,Z 831.58,A -85,B 0,C 180,E1 -17386.408,E2 -17386.408} C_VEL
LIN {X 0,Y 281.594,Z 823.374,A -85,B 0,C 180,E1 -17388.485,E2 -17388.485} C_VEL
LIN {X 0,Y 283.579,Z 814.415,A -85,B 0,C 180,E1 -17390.301,E2 -17390.301} C_VEL
LIN {X 0,Y 285.633,Z 804.98,A -85,B 0,C 180,E1 -17391.847,E2 -17391.847} C_VEL
LIN {X 0,Y 287.569,Z 794.822,A -85,B 0,C 180,E1 -17393.208,E2 -17393.208} C_VEL
LIN {X 0,Y 288.407,Z 784.06,A -85,B 0,C 180,E1 -17394.472,E2 -17394.472} C_VEL
LIN {X 0,Y 288.944,Z 771.393,A -85,B 0,C 180,E1 -17395.659,E2 -17395.659} C_VEL
LIN {X 0,Y 288.334,Z 760.772,A -85,B 0,C 180,E1 -17396.537,E2 -17396.537} C_VEL
LIN {X 0,Y 286.321,Z 748.313,A -85,B 0,C 180,E1 -17397.474,E2 -17397.474} C_VEL
LIN {X 0,Y 283.83,Z 737.353,A -85,B 0,C 180,E1 -17398.319,E2 -17398.319} C_VEL
LIN {X 0,Y 283.039,Z 722.3,A -85,B 0,C 180,E1 -17401.011,E2 -17401.011} C_VEL
